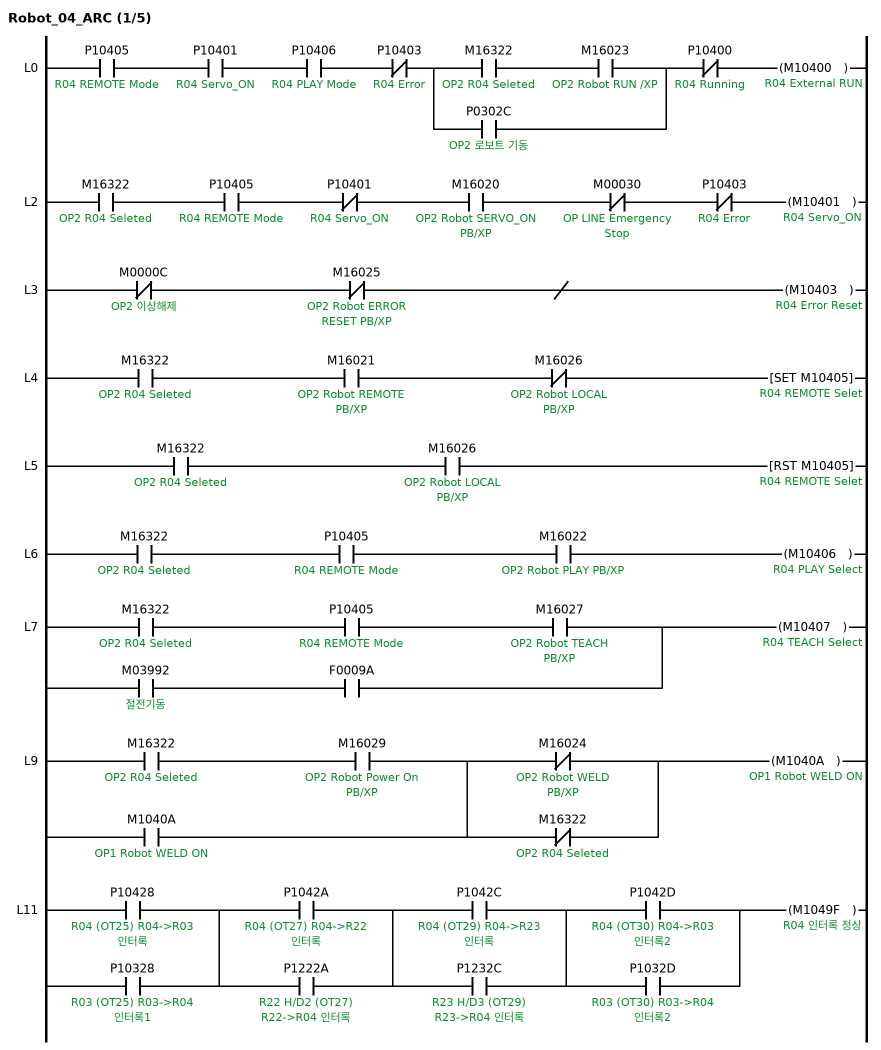
[picture p336: Robot_04_ARC rungs L0-L11]
; L0
LOAD      P10405	// R04 REMOTE Mode
AND       P10401	// R04 Servo_ON
AND       P10406	// R04 PLAY Mode
AND NOT   P10403	// R04 Error
LOAD      M16322	// OP2 R04 Seleted
AND       M16023	// OP2 Robot RUN /XP
OR        P0302C	// OP2 로보트 기동
AND LOAD
AND NOT   P10400	// R04 Running
OUT       M10400	// R04 External RUN
; L2
LOAD      M16322	// OP2 R04 Seleted
AND       P10405	// R04 REMOTE Mode
AND NOT   P10401	// R04 Servo_ON
AND       M16020	// OP2 Robot SERVO_ON PB/XP
AND NOT   M00030	// OP LINE Emergency Stop
AND NOT   P10403	// R04 Error
OUT       M10401	// R04 Servo_ON
; L3
LOAD NOT  M0000C	// OP2 이상해제
AND NOT   M16025	// OP2 Robot ERROR RESET PB/XP
NOT
OUT       M10403	// R04 Error Reset
; L4
LOAD      M16322	// OP2 R04 Seleted
AND       M16021	// OP2 Robot REMOTE PB/XP
AND NOT   M16026	// OP2 Robot LOCAL PB/XP
SET       M10405	// R04 REMOTE Selet
; L5
LOAD      M16322	// OP2 R04 Seleted
AND       M16026	// OP2 Robot LOCAL PB/XP
RST       M10405	// R04 REMOTE Selet
; L6
LOAD      M16322	// OP2 R04 Seleted
AND       P10405	// R04 REMOTE Mode
AND       M16022	// OP2 Robot PLAY PB/XP
OUT       M10406	// R04 PLAY Select
; L7
LOAD      M16322	// OP2 R04 Seleted
AND       P10405	// R04 REMOTE Mode
AND       M16027	// OP2 Robot TEACH PB/XP
LOAD      M03992	// 절전기동
AND       F0009A
OR LOAD
OUT       M10407	// R04 TEACH Select
; L9
LOAD      M16322	// OP2 R04 Seleted
AND       M16029	// OP2 Robot Power On PB/XP
OR        M1040A	// OP1 Robot WELD ON
LOAD NOT  M16024	// OP2 Robot WELD PB/XP
OR NOT    M16322	// OP2 R04 Seleted
AND LOAD
OUT       M1040A	// OP1 Robot WELD ON
; L11
LOAD      P10428	// R04 (OT25) R04->R03 인터록
OR        P10328	// R03 (OT25) R03->R04 인터록1
LOAD      P1042A	// R04 (OT27) R04->R22 인터록
OR        P1222A	// R22 H/D2 (OT27) R22->R04 인터록
AND LOAD
LOAD      P1042C	// R04 (OT29) R04->R23 인터록
OR        P1232C	// R23 H/D3 (OT29) R23->R04 인터록
AND LOAD
LOAD      P1042D	// R04 (OT30) R04->R03 인터록2
OR        P1032D	// R03 (OT30) R03->R04 인터록2
AND LOAD
OUT       M1049F	// R04 인터록 정상

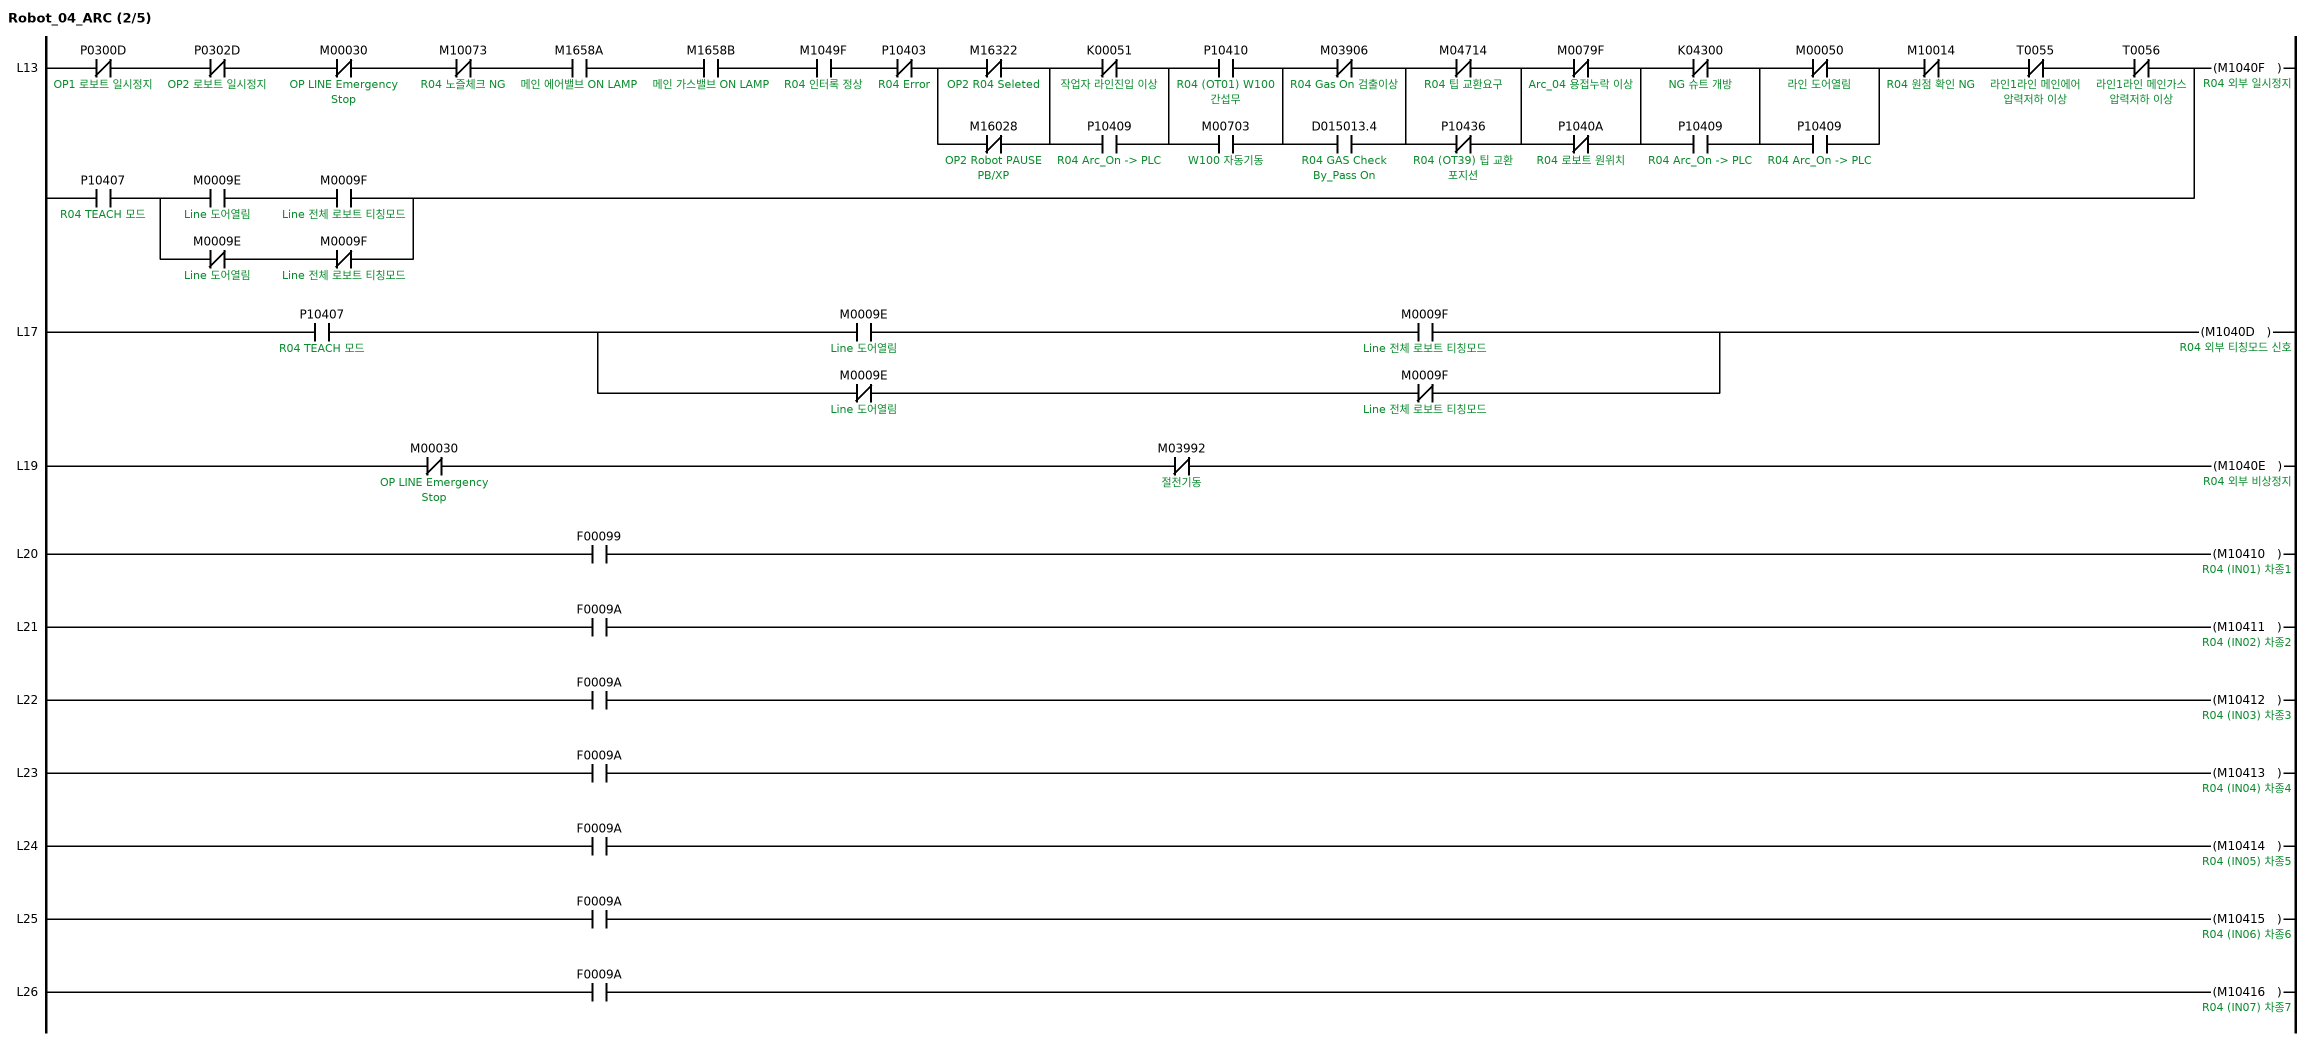
; L13
LOAD NOT  P0300D	// OP1 로보트 일시정지
AND NOT   P0302D	// OP2 로보트 일시정지
AND NOT   M00030	// OP LINE Emergency Stop
AND NOT   M10073	// R04 노즐체크 NG
AND       M1658A	// 메인 에어밸브 ON LAMP
AND       M1658B	// 메인 가스밸브 ON LAMP
AND       M1049F	// R04 인터록 정상
AND NOT   P10403	// R04 Error
LOAD NOT  M16322	// OP2 R04 Seleted
OR NOT    M16028	// OP2 Robot PAUSE PB/XP
AND LOAD
LOAD NOT  K00051	//  작업자 라인진입 이상
OR        P10409	// R04 Arc_On -> PLC
AND LOAD
LOAD      P10410	// R04 (OT01) W100 간섭무
OR        M00703	// W100 자동기동
AND LOAD
LOAD NOT  M03906	// R04 Gas On 검출이상
OR        D015013.4	// R04 GAS Check By_Pass On
AND LOAD
LOAD NOT  M04714	// R04 팁 교환요구
OR NOT    P10436	// R04 (OT39) 팁 교환 포지션
AND LOAD
LOAD NOT  M0079F	// Arc_04 용접누락 이상
OR NOT    P1040A	// R04 로보트 원위치
AND LOAD
LOAD NOT  K04300	// NG 슈트 개방
OR        P10409	// R04 Arc_On -> PLC
AND LOAD
LOAD NOT  M00050	// 라인 도어열림
OR        P10409	// R04 Arc_On -> PLC
AND LOAD
AND NOT   M10014	// R04 원점 확인 NG
AND NOT   T0055	// 라인1라인 메인에어 압력저하 이상
AND NOT   T0056	// 라인1라인 메인가스 압력저하 이상
LOAD      P10407	// R04 TEACH 모드
LOAD      M0009E	// Line 도어열림
AND       M0009F	// Line 전체 로보트 티칭모드
LOAD NOT  M0009E	// Line 도어열림
AND NOT   M0009F	// Line 전체 로보트 티칭모드
OR LOAD
AND LOAD
OR LOAD
OUT       M1040F	// R04 외부 일시정지
; L17
LOAD      P10407	// R04 TEACH 모드
LOAD      M0009E	// Line 도어열림
AND       M0009F	// Line 전체 로보트 티칭모드
LOAD NOT  M0009E	// Line 도어열림
AND NOT   M0009F	// Line 전체 로보트 티칭모드
OR LOAD
AND LOAD
OUT       M1040D	// R04 외부 티칭모드 신호
; L19
LOAD NOT  M00030	// OP LINE Emergency Stop
AND NOT   M03992	// 절전기동
OUT       M1040E	// R04 외부 비상정지 
; L20
LOAD      F00099
OUT       M10410	// R04 (IN01) 차종1
; L21
LOAD      F0009A
OUT       M10411	// R04 (IN02) 차종2
; L22
LOAD      F0009A
OUT       M10412	// R04 (IN03) 차종3
; L23
LOAD      F0009A
OUT       M10413	// R04 (IN04) 차종4
; L24
LOAD      F0009A
OUT       M10414	// R04 (IN05) 차종5
; L25
LOAD      F0009A
OUT       M10415	// R04 (IN06) 차종6
; L26
LOAD      F0009A
OUT       M10416	// R04 (IN07) 차종7

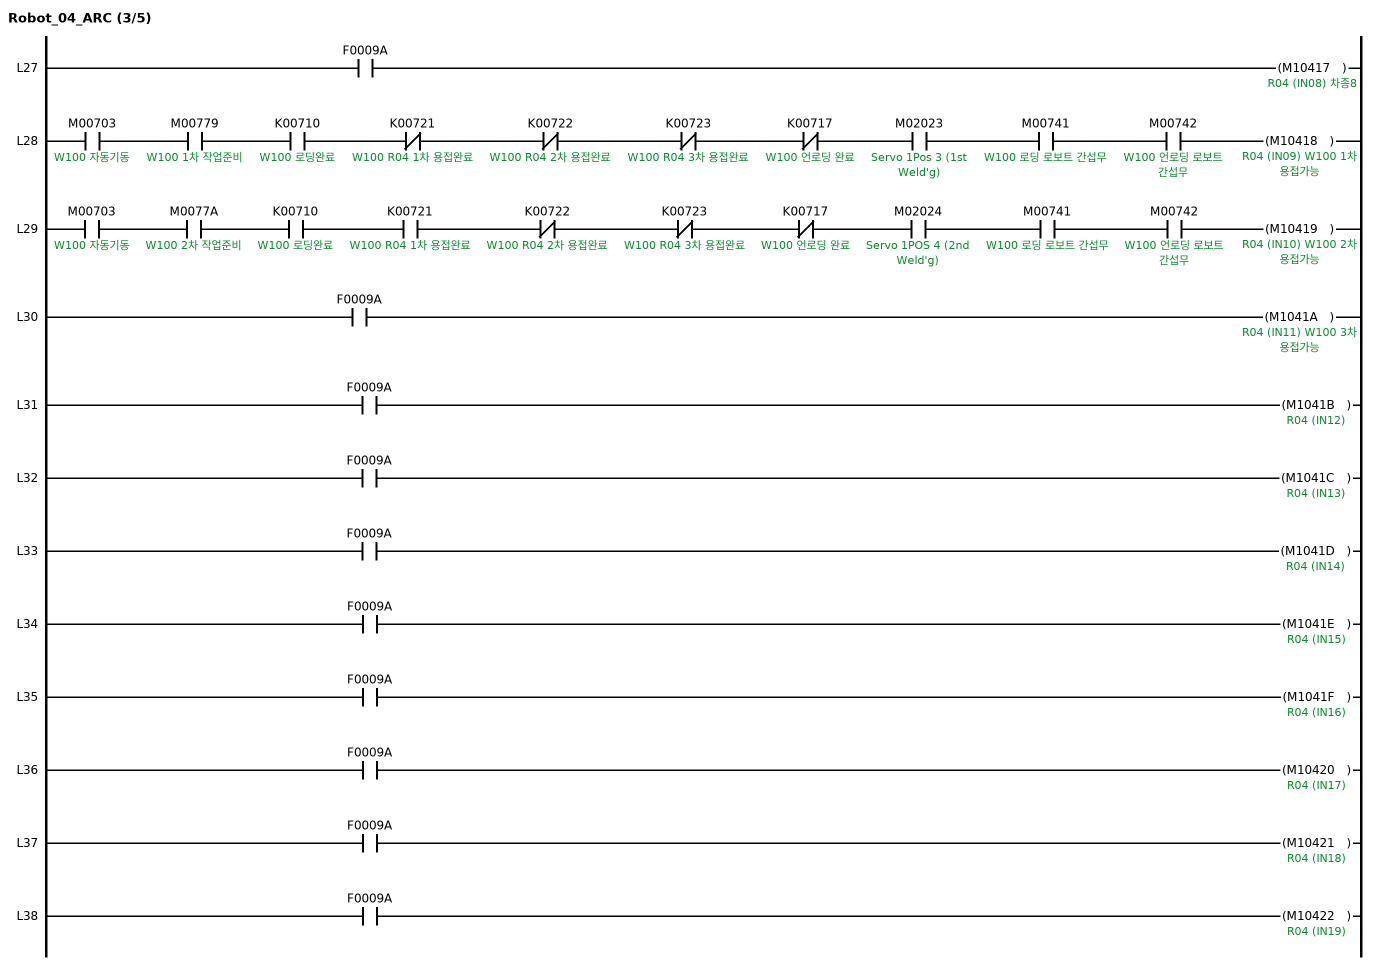
; L27
LOAD      F0009A
OUT       M10417	// R04 (IN08) 차종8
; L28
LOAD      M00703	// W100 자동기동
AND       M00779	// W100 1차 작업준비
AND       K00710	// W100 로딩완료
AND NOT   K00721	// W100 R04 1차 용접완료
AND NOT   K00722	// W100 R04 2차 용접완료
AND NOT   K00723	// W100 R04 3차 용접완료
AND NOT   K00717	// W100 언로딩 완료
AND       M02023	// Servo 1Pos 3 (1st Weld'g)
AND       M00741	// W100 로딩 로보트 간섭무
AND       M00742	// W100 언로딩 로보트 간섭무
OUT       M10418	// R04 (IN09) W100 1차 용접가능
; L29
LOAD      M00703	// W100 자동기동
AND       M0077A	// W100 2차 작업준비
AND       K00710	// W100 로딩완료
AND       K00721	// W100 R04 1차 용접완료
AND NOT   K00722	// W100 R04 2차 용접완료
AND NOT   K00723	// W100 R04 3차 용접완료
AND NOT   K00717	// W100 언로딩 완료
AND       M02024	// Servo 1POS 4 (2nd Weld'g)
AND       M00741	// W100 로딩 로보트 간섭무
AND       M00742	// W100 언로딩 로보트 간섭무
OUT       M10419	// R04 (IN10) W100 2차 용접가능
; L30
LOAD      F0009A
OUT       M1041A	// R04 (IN11) W100 3차 용접가능
; L31
LOAD      F0009A
OUT       M1041B	// R04 (IN12)
; L32
LOAD      F0009A
OUT       M1041C	// R04 (IN13)
; L33
LOAD      F0009A
OUT       M1041D	// R04 (IN14)
; L34
LOAD      F0009A
OUT       M1041E	// R04 (IN15)
; L35
LOAD      F0009A
OUT       M1041F	// R04 (IN16)
; L36
LOAD      F0009A
OUT       M10420	// R04 (IN17)
; L37
LOAD      F0009A
OUT       M10421	// R04 (IN18)
; L38
LOAD      F0009A
OUT       M10422	// R04 (IN19)

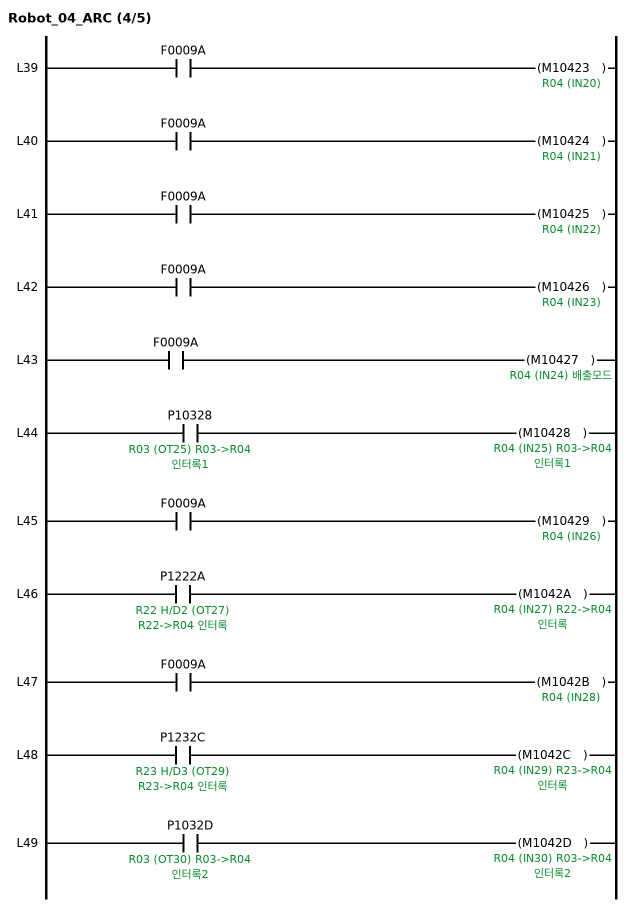
; L39
LOAD      F0009A
OUT       M10423	// R04 (IN20)
; L40
LOAD      F0009A
OUT       M10424	// R04 (IN21)
; L41
LOAD      F0009A
OUT       M10425	// R04 (IN22)
; L42
LOAD      F0009A
OUT       M10426	// R04 (IN23)
; L43
LOAD      F0009A
OUT       M10427	// R04 (IN24) 배출모드
; L44
LOAD      P10328	// R03 (OT25) R03->R04 인터록1
OUT       M10428	// R04 (IN25) R03->R04 인터록1
; L45
LOAD      F0009A
OUT       M10429	// R04 (IN26)
; L46
LOAD      P1222A	// R22 H/D2 (OT27) R22->R04 인터록
OUT       M1042A	// R04 (IN27) R22->R04 인터록
; L47
LOAD      F0009A
OUT       M1042B	// R04 (IN28)
; L48
LOAD      P1232C	// R23 H/D3 (OT29) R23->R04 인터록
OUT       M1042C	// R04 (IN29) R23->R04 인터록
; L49
LOAD      P1032D	// R03 (OT30) R03->R04 인터록2
OUT       M1042D	// R04 (IN30) R03->R04 인터록2

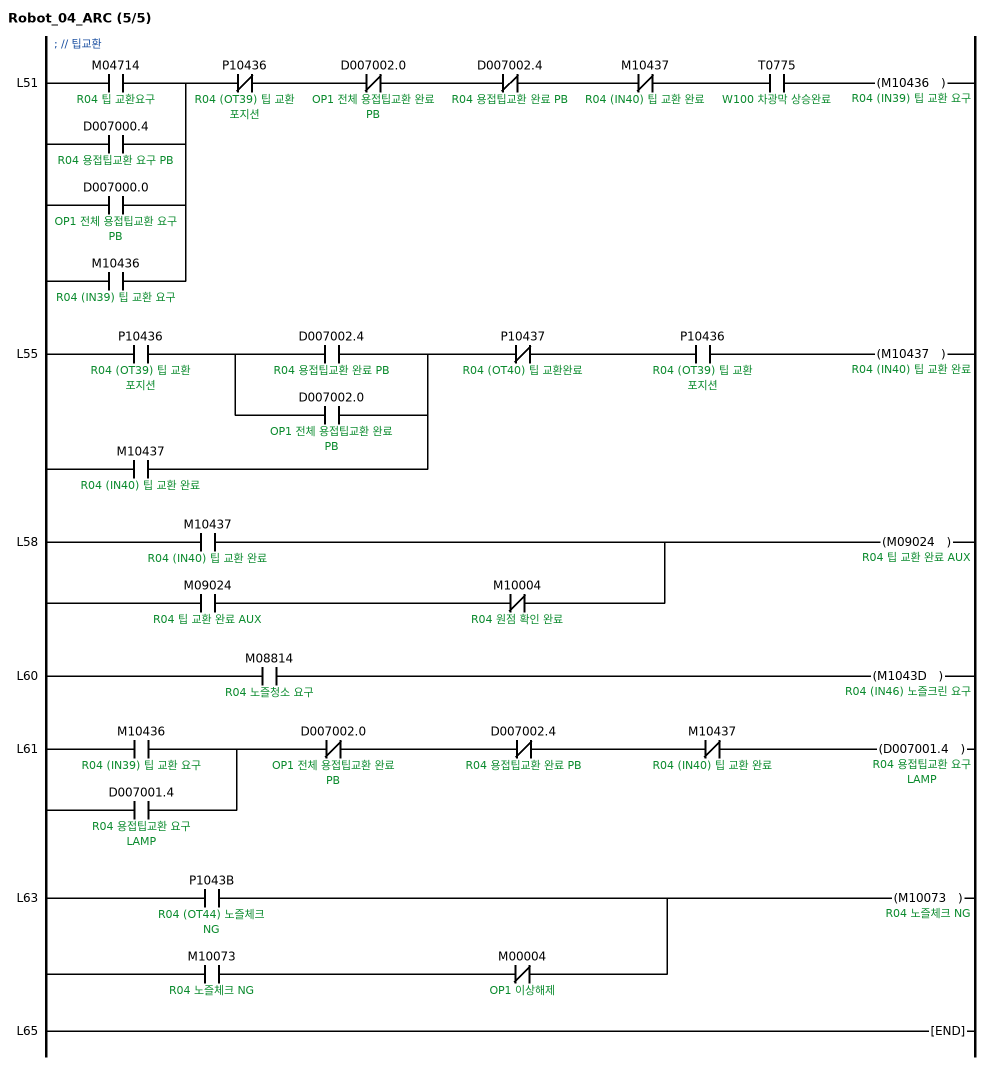
//  // 팁교환
; L51
LOAD      M04714	// R04 팁 교환요구
OR        D007000.4	// R04 용접팁교환 요구 PB
OR        D007000.0	// OP1 전체 용접팁교환 요구 PB
OR        M10436	// R04 (IN39) 팁 교환 요구
AND NOT   P10436	// R04 (OT39) 팁 교환 포지션
AND NOT   D007002.0	// OP1 전체 용접팁교환 완료 PB
AND NOT   D007002.4	// R04 용접팁교환 완료 PB
AND NOT   M10437	// R04 (IN40) 팁 교환 완료
AND       T0775	// W100 차광막 상승완료
OUT       M10436	// R04 (IN39) 팁 교환 요구
; L55
LOAD      P10436	// R04 (OT39) 팁 교환 포지션
LOAD      D007002.4	// R04 용접팁교환 완료 PB
OR        D007002.0	// OP1 전체 용접팁교환 완료 PB
AND LOAD
OR        M10437	// R04 (IN40) 팁 교환 완료
AND NOT   P10437	// R04 (OT40) 팁 교환완료
AND       P10436	// R04 (OT39) 팁 교환 포지션
OUT       M10437	// R04 (IN40) 팁 교환 완료
; L58
LOAD      M10437	// R04 (IN40) 팁 교환 완료
LOAD      M09024	// R04 팁 교환 완료 AUX
AND NOT   M10004	// R04 원점 확인 완료
OR LOAD
OUT       M09024	// R04 팁 교환 완료 AUX
; L60
LOAD      M08814	// R04 노즐청소 요구
OUT       M1043D	// R04 (IN46) 노즐크린 요구
; L61
LOAD      M10436	// R04 (IN39) 팁 교환 요구
OR        D007001.4	// R04 용접팁교환 요구 LAMP
AND NOT   D007002.0	// OP1 전체 용접팁교환 완료 PB
AND NOT   D007002.4	// R04 용접팁교환 완료 PB
AND NOT   M10437	// R04 (IN40) 팁 교환 완료
OUT       D007001.4	// R04 용접팁교환 요구 LAMP
; L63
LOAD      P1043B	// R04 (OT44) 노즐체크 NG
LOAD      M10073	// R04 노즐체크 NG
AND NOT   M00004	// OP1 이상해제
OR LOAD
OUT       M10073	// R04 노즐체크 NG
; L65
END

PROGRAM Robot_05_ARC (task: 스캔 프로그램)

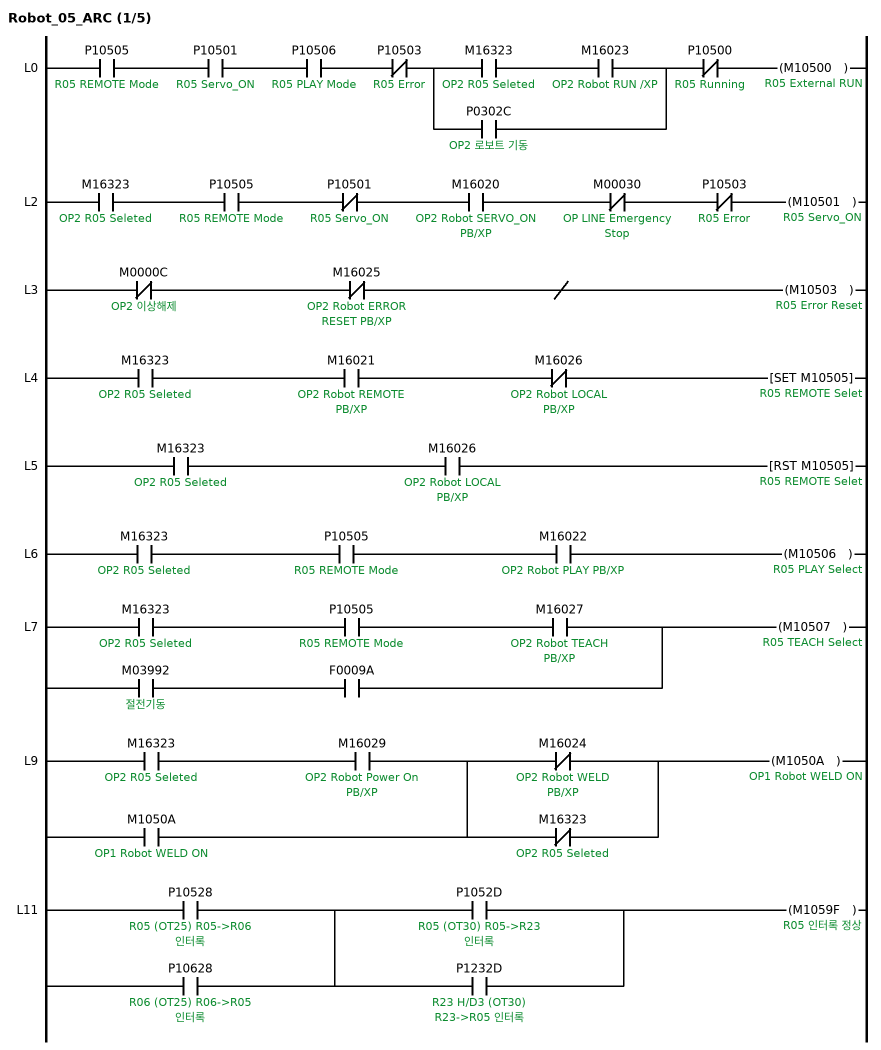
; L0
LOAD      P10505	// R05 REMOTE Mode
AND       P10501	// R05 Servo_ON
AND       P10506	// R05 PLAY Mode
AND NOT   P10503	// R05 Error
LOAD      M16323	// OP2 R05 Seleted
AND       M16023	// OP2 Robot RUN /XP
OR        P0302C	// OP2 로보트 기동
AND LOAD
AND NOT   P10500	// R05 Running
OUT       M10500	// R05 External RUN
; L2
LOAD      M16323	// OP2 R05 Seleted
AND       P10505	// R05 REMOTE Mode
AND NOT   P10501	// R05 Servo_ON
AND       M16020	// OP2 Robot SERVO_ON PB/XP
AND NOT   M00030	// OP LINE Emergency Stop
AND NOT   P10503	// R05 Error
OUT       M10501	// R05 Servo_ON
; L3
LOAD NOT  M0000C	// OP2 이상해제
AND NOT   M16025	// OP2 Robot ERROR RESET PB/XP
NOT
OUT       M10503	// R05 Error Reset
; L4
LOAD      M16323	// OP2 R05 Seleted
AND       M16021	// OP2 Robot REMOTE PB/XP
AND NOT   M16026	// OP2 Robot LOCAL PB/XP
SET       M10505	// R05 REMOTE Selet
; L5
LOAD      M16323	// OP2 R05 Seleted
AND       M16026	// OP2 Robot LOCAL PB/XP
RST       M10505	// R05 REMOTE Selet
; L6
LOAD      M16323	// OP2 R05 Seleted
AND       P10505	// R05 REMOTE Mode
AND       M16022	// OP2 Robot PLAY PB/XP
OUT       M10506	// R05 PLAY Select
; L7
LOAD      M16323	// OP2 R05 Seleted
AND       P10505	// R05 REMOTE Mode
AND       M16027	// OP2 Robot TEACH PB/XP
LOAD      M03992	// 절전기동
AND       F0009A
OR LOAD
OUT       M10507	// R05 TEACH Select
; L9
LOAD      M16323	// OP2 R05 Seleted
AND       M16029	// OP2 Robot Power On PB/XP
OR        M1050A	// OP1 Robot WELD ON
LOAD NOT  M16024	// OP2 Robot WELD PB/XP
OR NOT    M16323	// OP2 R05 Seleted
AND LOAD
OUT       M1050A	// OP1 Robot WELD ON
; L11
LOAD      P10528	// R05 (OT25) R05->R06 인터록
OR        P10628	// R06 (OT25) R06->R05 인터록
LOAD      P1052D	// R05 (OT30) R05->R23 인터록
OR        P1232D	// R23 H/D3 (OT30) R23->R05 인터록
AND LOAD
OUT       M1059F	// R05 인터록 정상

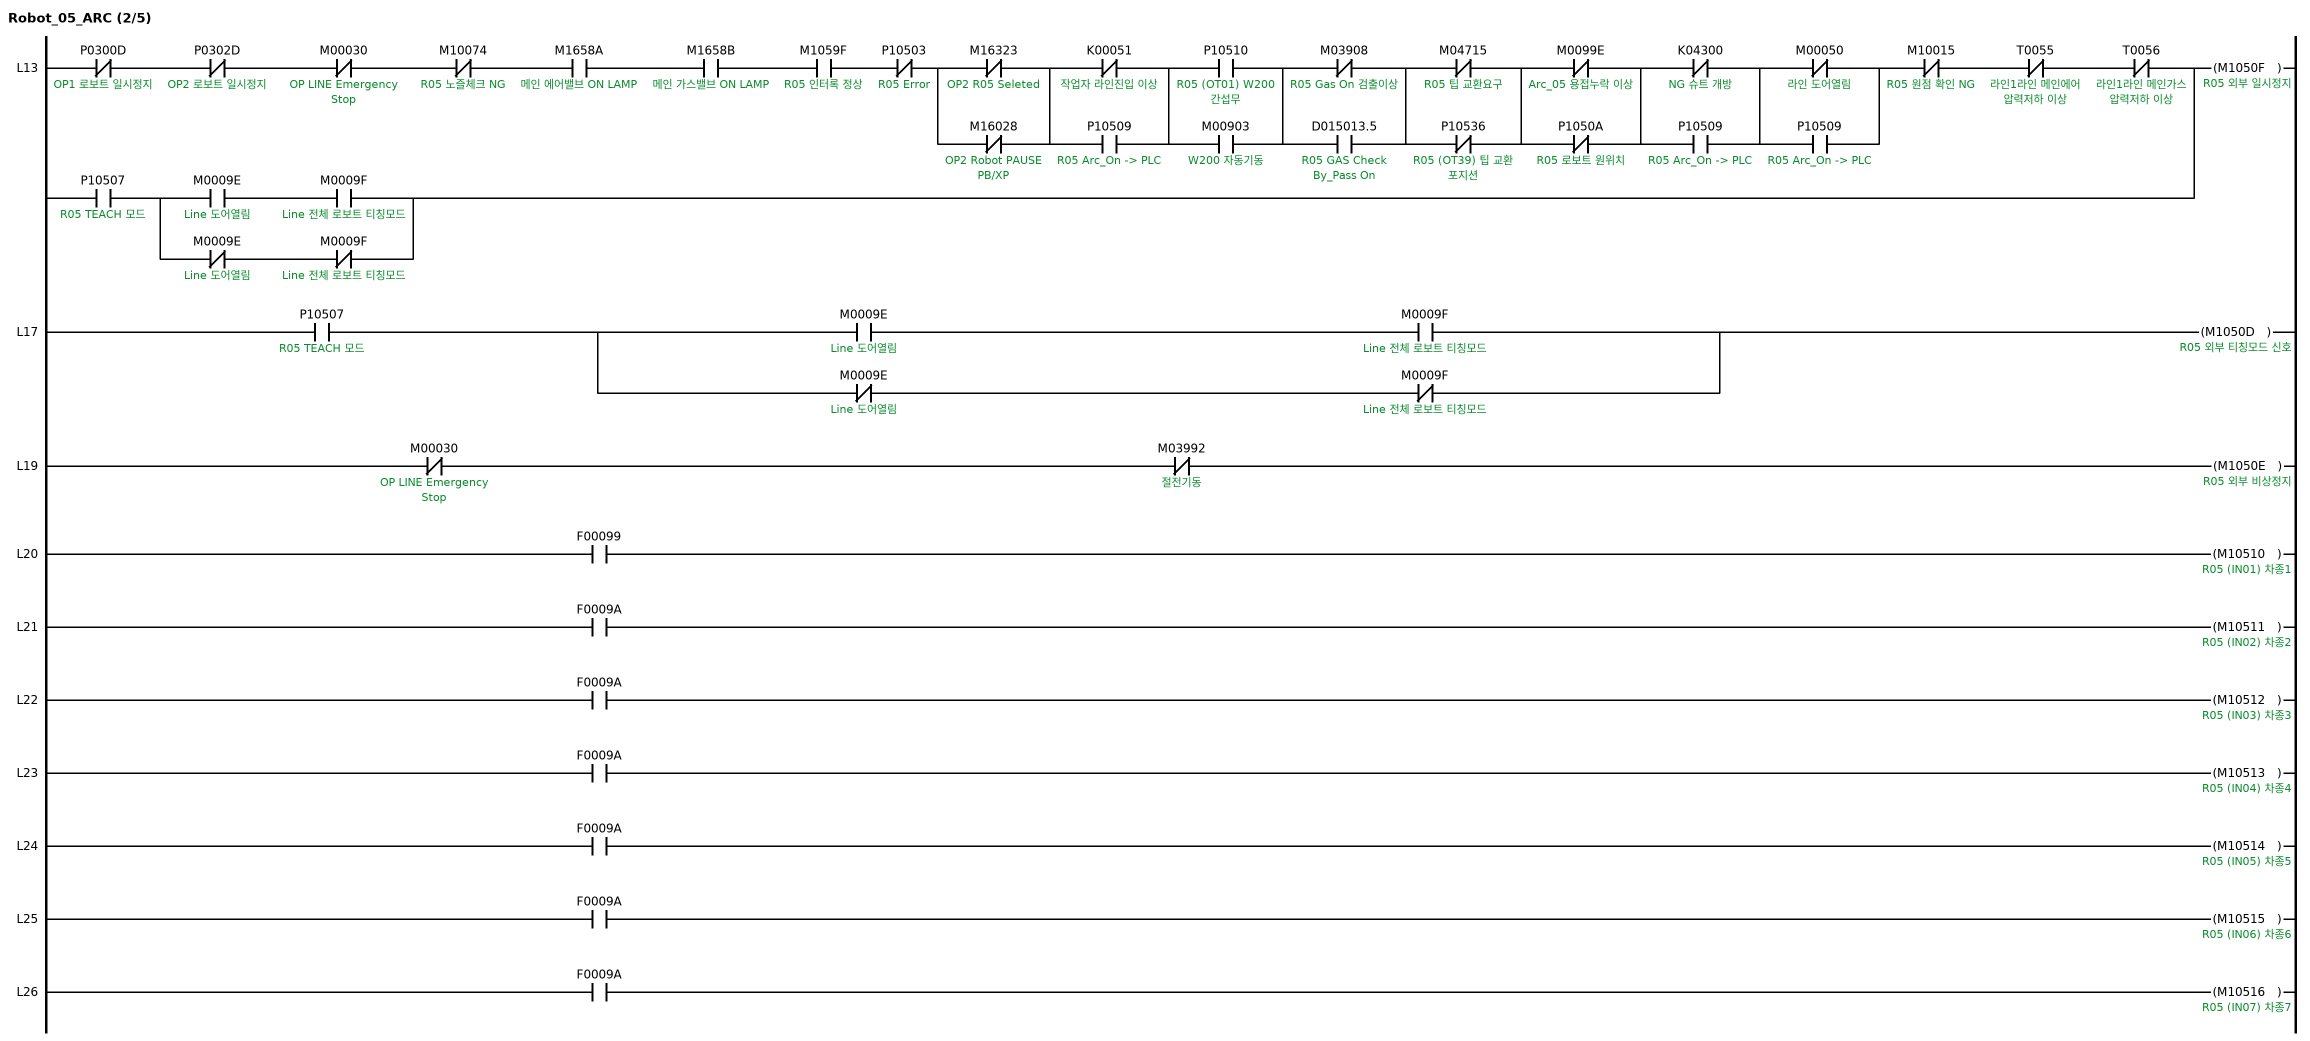
; L13
LOAD NOT  P0300D	// OP1 로보트 일시정지
AND NOT   P0302D	// OP2 로보트 일시정지
AND NOT   M00030	// OP LINE Emergency Stop
AND NOT   M10074	// R05 노즐체크 NG
AND       M1658A	// 메인 에어밸브 ON LAMP
AND       M1658B	// 메인 가스밸브 ON LAMP
AND       M1059F	// R05 인터록 정상
AND NOT   P10503	// R05 Error
LOAD NOT  M16323	// OP2 R05 Seleted
OR NOT    M16028	// OP2 Robot PAUSE PB/XP
AND LOAD
LOAD NOT  K00051	//  작업자 라인진입 이상
OR        P10509	// R05 Arc_On -> PLC
AND LOAD
LOAD      P10510	// R05 (OT01) W200 간섭무
OR        M00903	// W200 자동기동
AND LOAD
LOAD NOT  M03908	// R05 Gas On 검출이상
OR        D015013.5	// R05 GAS Check By_Pass On
AND LOAD
LOAD NOT  M04715	// R05 팁 교환요구
OR NOT    P10536	// R05 (OT39) 팁 교환 포지션
AND LOAD
LOAD NOT  M0099E	// Arc_05 용접누락 이상
OR NOT    P1050A	// R05 로보트 원위치
AND LOAD
LOAD NOT  K04300	// NG 슈트 개방
OR        P10509	// R05 Arc_On -> PLC
AND LOAD
LOAD NOT  M00050	// 라인 도어열림
OR        P10509	// R05 Arc_On -> PLC
AND LOAD
AND NOT   M10015	// R05 원점 확인 NG
AND NOT   T0055	// 라인1라인 메인에어 압력저하 이상
AND NOT   T0056	// 라인1라인 메인가스 압력저하 이상
LOAD      P10507	// R05 TEACH 모드
LOAD      M0009E	// Line 도어열림
AND       M0009F	// Line 전체 로보트 티칭모드
LOAD NOT  M0009E	// Line 도어열림
AND NOT   M0009F	// Line 전체 로보트 티칭모드
OR LOAD
AND LOAD
OR LOAD
OUT       M1050F	// R05 외부 일시정지
; L17
LOAD      P10507	// R05 TEACH 모드
LOAD      M0009E	// Line 도어열림
AND       M0009F	// Line 전체 로보트 티칭모드
LOAD NOT  M0009E	// Line 도어열림
AND NOT   M0009F	// Line 전체 로보트 티칭모드
OR LOAD
AND LOAD
OUT       M1050D	// R05 외부 티칭모드 신호
; L19
LOAD NOT  M00030	// OP LINE Emergency Stop
AND NOT   M03992	// 절전기동
OUT       M1050E	// R05 외부 비상정지 
; L20
LOAD      F00099
OUT       M10510	// R05 (IN01) 차종1
; L21
LOAD      F0009A
OUT       M10511	// R05 (IN02) 차종2
; L22
LOAD      F0009A
OUT       M10512	// R05 (IN03) 차종3
; L23
LOAD      F0009A
OUT       M10513	// R05 (IN04) 차종4
; L24
LOAD      F0009A
OUT       M10514	// R05 (IN05) 차종5
; L25
LOAD      F0009A
OUT       M10515	// R05 (IN06) 차종6
; L26
LOAD      F0009A
OUT       M10516	// R05 (IN07) 차종7

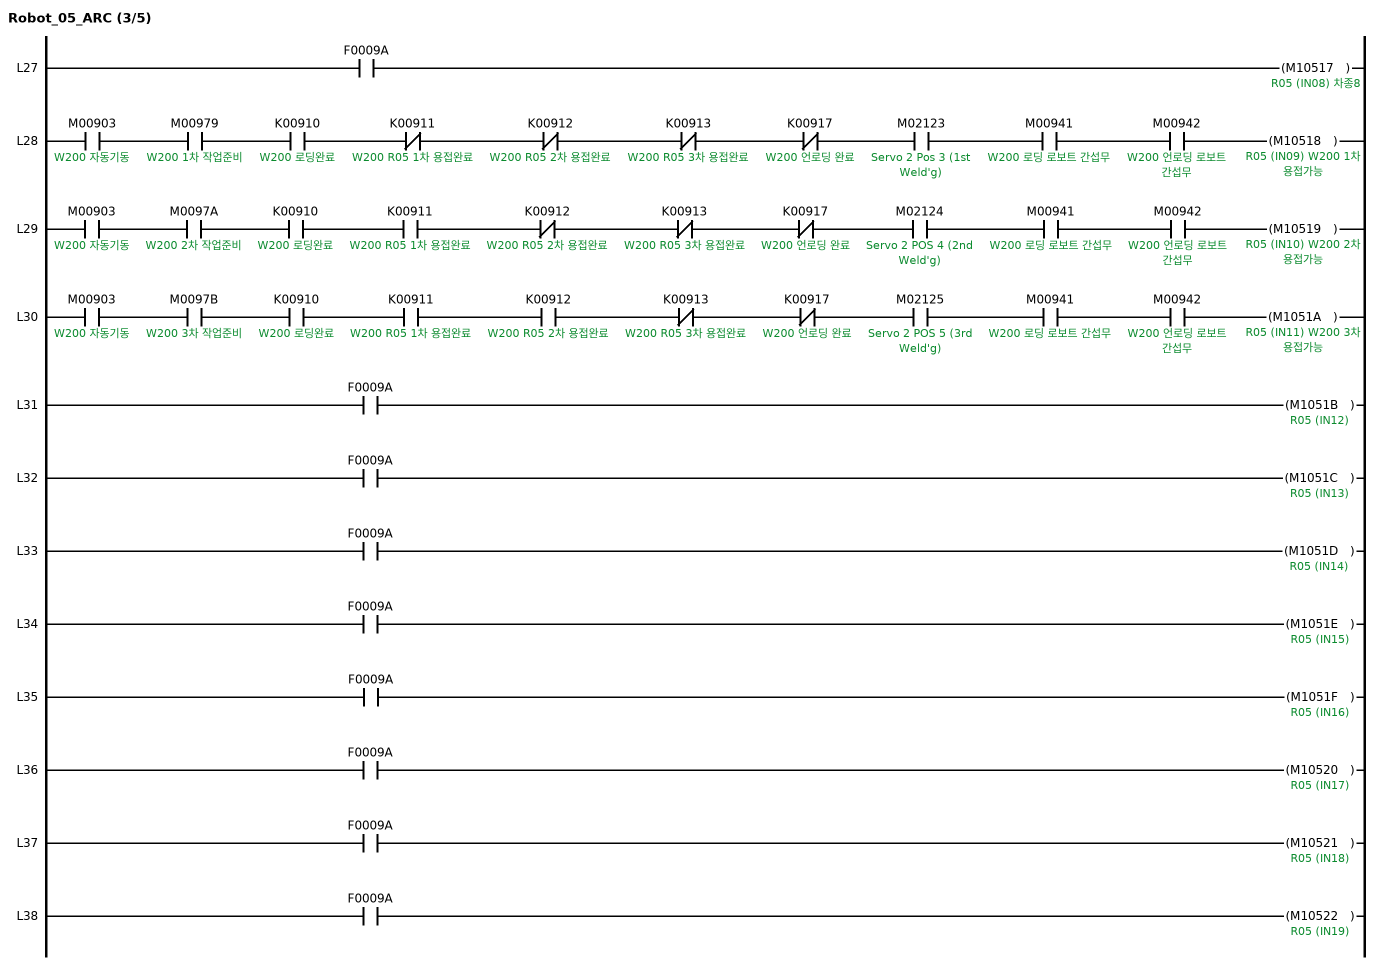
; L27
LOAD      F0009A
OUT       M10517	// R05 (IN08) 차종8
; L28
LOAD      M00903	// W200 자동기동
AND       M00979	// W200 1차 작업준비
AND       K00910	// W200 로딩완료
AND NOT   K00911	// W200 R05 1차 용접완료
AND NOT   K00912	// W200 R05 2차 용접완료
AND NOT   K00913	// W200 R05 3차 용접완료
AND NOT   K00917	// W200 언로딩 완료
AND       M02123	// Servo 2 Pos 3 (1st Weld'g)
AND       M00941	// W200 로딩 로보트 간섭무
AND       M00942	// W200 언로딩 로보트 간섭무
OUT       M10518	// R05 (IN09) W200 1차 용접가능
; L29
LOAD      M00903	// W200 자동기동
AND       M0097A	// W200 2차 작업준비
AND       K00910	// W200 로딩완료
AND       K00911	// W200 R05 1차 용접완료
AND NOT   K00912	// W200 R05 2차 용접완료
AND NOT   K00913	// W200 R05 3차 용접완료
AND NOT   K00917	// W200 언로딩 완료
AND       M02124	// Servo 2 POS 4 (2nd Weld'g)
AND       M00941	// W200 로딩 로보트 간섭무
AND       M00942	// W200 언로딩 로보트 간섭무
OUT       M10519	// R05 (IN10) W200 2차 용접가능
; L30
LOAD      M00903	// W200 자동기동
AND       M0097B	// W200 3차 작업준비
AND       K00910	// W200 로딩완료
AND       K00911	// W200 R05 1차 용접완료
AND       K00912	// W200 R05 2차 용접완료
AND NOT   K00913	// W200 R05 3차 용접완료
AND NOT   K00917	// W200 언로딩 완료
AND       M02125	// Servo 2 POS 5 (3rd Weld'g)
AND       M00941	// W200 로딩 로보트 간섭무
AND       M00942	// W200 언로딩 로보트 간섭무
OUT       M1051A	// R05 (IN11) W200 3차 용접가능
; L31
LOAD      F0009A
OUT       M1051B	// R05 (IN12)
; L32
LOAD      F0009A
OUT       M1051C	// R05 (IN13)
; L33
LOAD      F0009A
OUT       M1051D	// R05 (IN14)
; L34
LOAD      F0009A
OUT       M1051E	// R05 (IN15)
; L35
LOAD      F0009A
OUT       M1051F	// R05 (IN16)
; L36
LOAD      F0009A
OUT       M10520	// R05 (IN17)
; L37
LOAD      F0009A
OUT       M10521	// R05 (IN18)
; L38
LOAD      F0009A
OUT       M10522	// R05 (IN19)

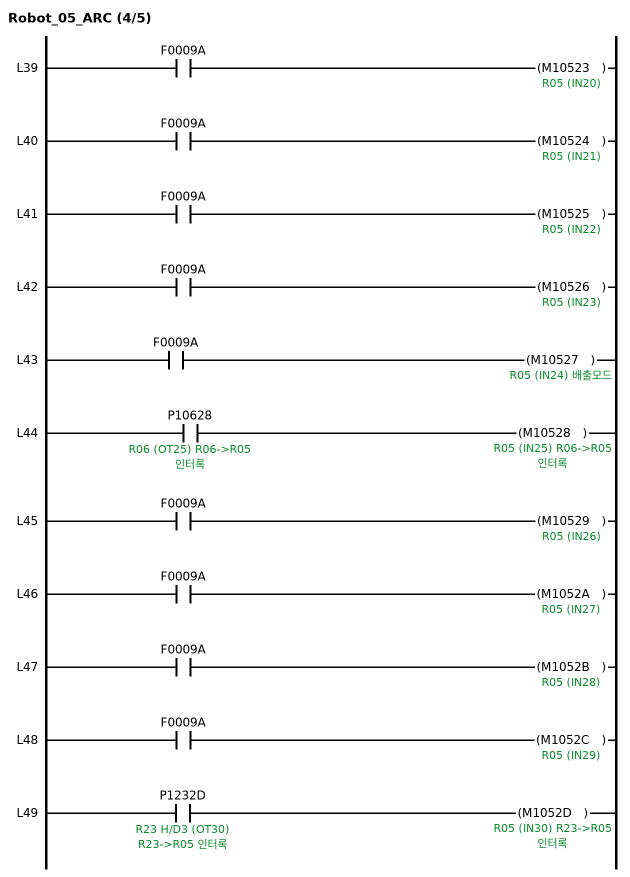
; L39
LOAD      F0009A
OUT       M10523	// R05 (IN20)
; L40
LOAD      F0009A
OUT       M10524	// R05 (IN21)
; L41
LOAD      F0009A
OUT       M10525	// R05 (IN22)
; L42
LOAD      F0009A
OUT       M10526	// R05 (IN23)
; L43
LOAD      F0009A
OUT       M10527	// R05 (IN24) 배출모드
; L44
LOAD      P10628	// R06 (OT25) R06->R05 인터록
OUT       M10528	// R05 (IN25) R06->R05 인터록
; L45
LOAD      F0009A
OUT       M10529	// R05 (IN26)
; L46
LOAD      F0009A
OUT       M1052A	// R05 (IN27)
; L47
LOAD      F0009A
OUT       M1052B	// R05 (IN28)
; L48
LOAD      F0009A
OUT       M1052C	// R05 (IN29)
; L49
LOAD      P1232D	// R23 H/D3 (OT30) R23->R05 인터록
OUT       M1052D	// R05 (IN30) R23->R05 인터록

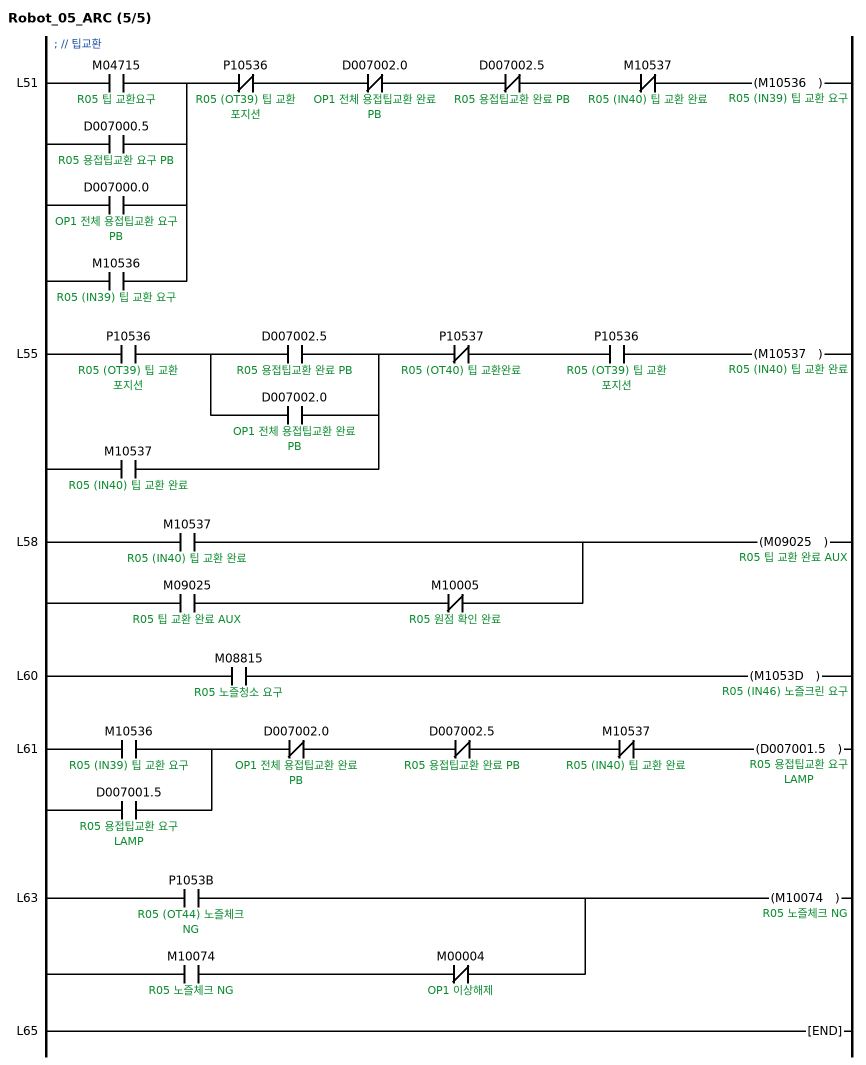
//  // 팁교환
; L51
LOAD      M04715	// R05 팁 교환요구
OR        D007000.5	// R05 용접팁교환 요구 PB
OR        D007000.0	// OP1 전체 용접팁교환 요구 PB
OR        M10536	// R05 (IN39) 팁 교환 요구
AND NOT   P10536	// R05 (OT39) 팁 교환 포지션
AND NOT   D007002.0	// OP1 전체 용접팁교환 완료 PB
AND NOT   D007002.5	// R05 용접팁교환 완료 PB
AND NOT   M10537	// R05 (IN40) 팁 교환 완료
OUT       M10536	// R05 (IN39) 팁 교환 요구
; L55
LOAD      P10536	// R05 (OT39) 팁 교환 포지션
LOAD      D007002.5	// R05 용접팁교환 완료 PB
OR        D007002.0	// OP1 전체 용접팁교환 완료 PB
AND LOAD
OR        M10537	// R05 (IN40) 팁 교환 완료
AND NOT   P10537	// R05 (OT40) 팁 교환완료
AND       P10536	// R05 (OT39) 팁 교환 포지션
OUT       M10537	// R05 (IN40) 팁 교환 완료
; L58
LOAD      M10537	// R05 (IN40) 팁 교환 완료
LOAD      M09025	// R05 팁 교환 완료 AUX
AND NOT   M10005	// R05 원점 확인 완료
OR LOAD
OUT       M09025	// R05 팁 교환 완료 AUX
; L60
LOAD      M08815	// R05 노즐청소 요구
OUT       M1053D	// R05 (IN46) 노즐크린 요구
; L61
LOAD      M10536	// R05 (IN39) 팁 교환 요구
OR        D007001.5	// R05 용접팁교환 요구 LAMP
AND NOT   D007002.0	// OP1 전체 용접팁교환 완료 PB
AND NOT   D007002.5	// R05 용접팁교환 완료 PB
AND NOT   M10537	// R05 (IN40) 팁 교환 완료
OUT       D007001.5	// R05 용접팁교환 요구 LAMP
; L63
LOAD      P1053B	// R05 (OT44) 노즐체크 NG
LOAD      M10074	// R05 노즐체크 NG
AND NOT   M00004	// OP1 이상해제
OR LOAD
OUT       M10074	// R05 노즐체크 NG
; L65
END

PROGRAM Robot_06_ARC (task: 스캔 프로그램)

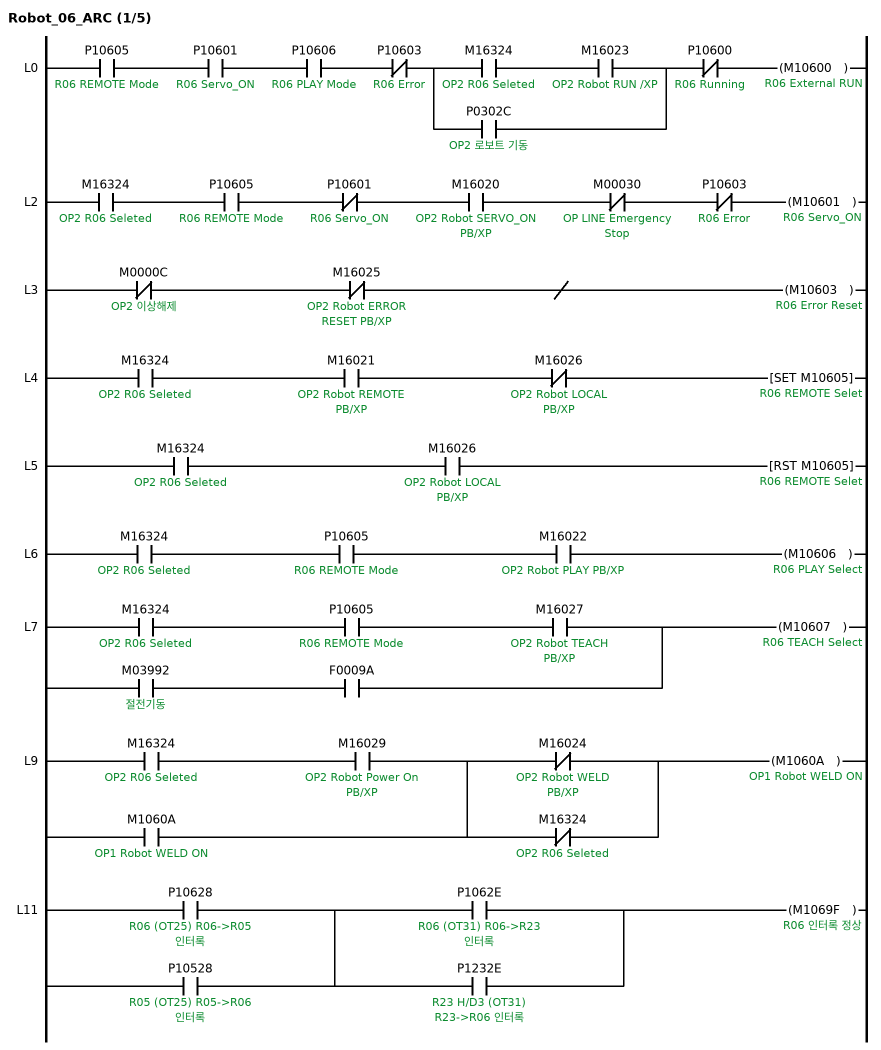
; L0
LOAD      P10605	// R06 REMOTE Mode
AND       P10601	// R06 Servo_ON
AND       P10606	// R06 PLAY Mode
AND NOT   P10603	// R06 Error
LOAD      M16324	// OP2 R06 Seleted
AND       M16023	// OP2 Robot RUN /XP
OR        P0302C	// OP2 로보트 기동
AND LOAD
AND NOT   P10600	// R06 Running
OUT       M10600	// R06 External RUN
; L2
LOAD      M16324	// OP2 R06 Seleted
AND       P10605	// R06 REMOTE Mode
AND NOT   P10601	// R06 Servo_ON
AND       M16020	// OP2 Robot SERVO_ON PB/XP
AND NOT   M00030	// OP LINE Emergency Stop
AND NOT   P10603	// R06 Error
OUT       M10601	// R06 Servo_ON
; L3
LOAD NOT  M0000C	// OP2 이상해제
AND NOT   M16025	// OP2 Robot ERROR RESET PB/XP
NOT
OUT       M10603	// R06 Error Reset
; L4
LOAD      M16324	// OP2 R06 Seleted
AND       M16021	// OP2 Robot REMOTE PB/XP
AND NOT   M16026	// OP2 Robot LOCAL PB/XP
SET       M10605	// R06 REMOTE Selet
; L5
LOAD      M16324	// OP2 R06 Seleted
AND       M16026	// OP2 Robot LOCAL PB/XP
RST       M10605	// R06 REMOTE Selet
; L6
LOAD      M16324	// OP2 R06 Seleted
AND       P10605	// R06 REMOTE Mode
AND       M16022	// OP2 Robot PLAY PB/XP
OUT       M10606	// R06 PLAY Select
; L7
LOAD      M16324	// OP2 R06 Seleted
AND       P10605	// R06 REMOTE Mode
AND       M16027	// OP2 Robot TEACH PB/XP
LOAD      M03992	// 절전기동
AND       F0009A
OR LOAD
OUT       M10607	// R06 TEACH Select
; L9
LOAD      M16324	// OP2 R06 Seleted
AND       M16029	// OP2 Robot Power On PB/XP
OR        M1060A	// OP1 Robot WELD ON
LOAD NOT  M16024	// OP2 Robot WELD PB/XP
OR NOT    M16324	// OP2 R06 Seleted
AND LOAD
OUT       M1060A	// OP1 Robot WELD ON
; L11
LOAD      P10628	// R06 (OT25) R06->R05 인터록
OR        P10528	// R05 (OT25) R05->R06 인터록
LOAD      P1062E	// R06 (OT31) R06->R23 인터록
OR        P1232E	// R23 H/D3 (OT31) R23->R06 인터록
AND LOAD
OUT       M1069F	// R06 인터록 정상

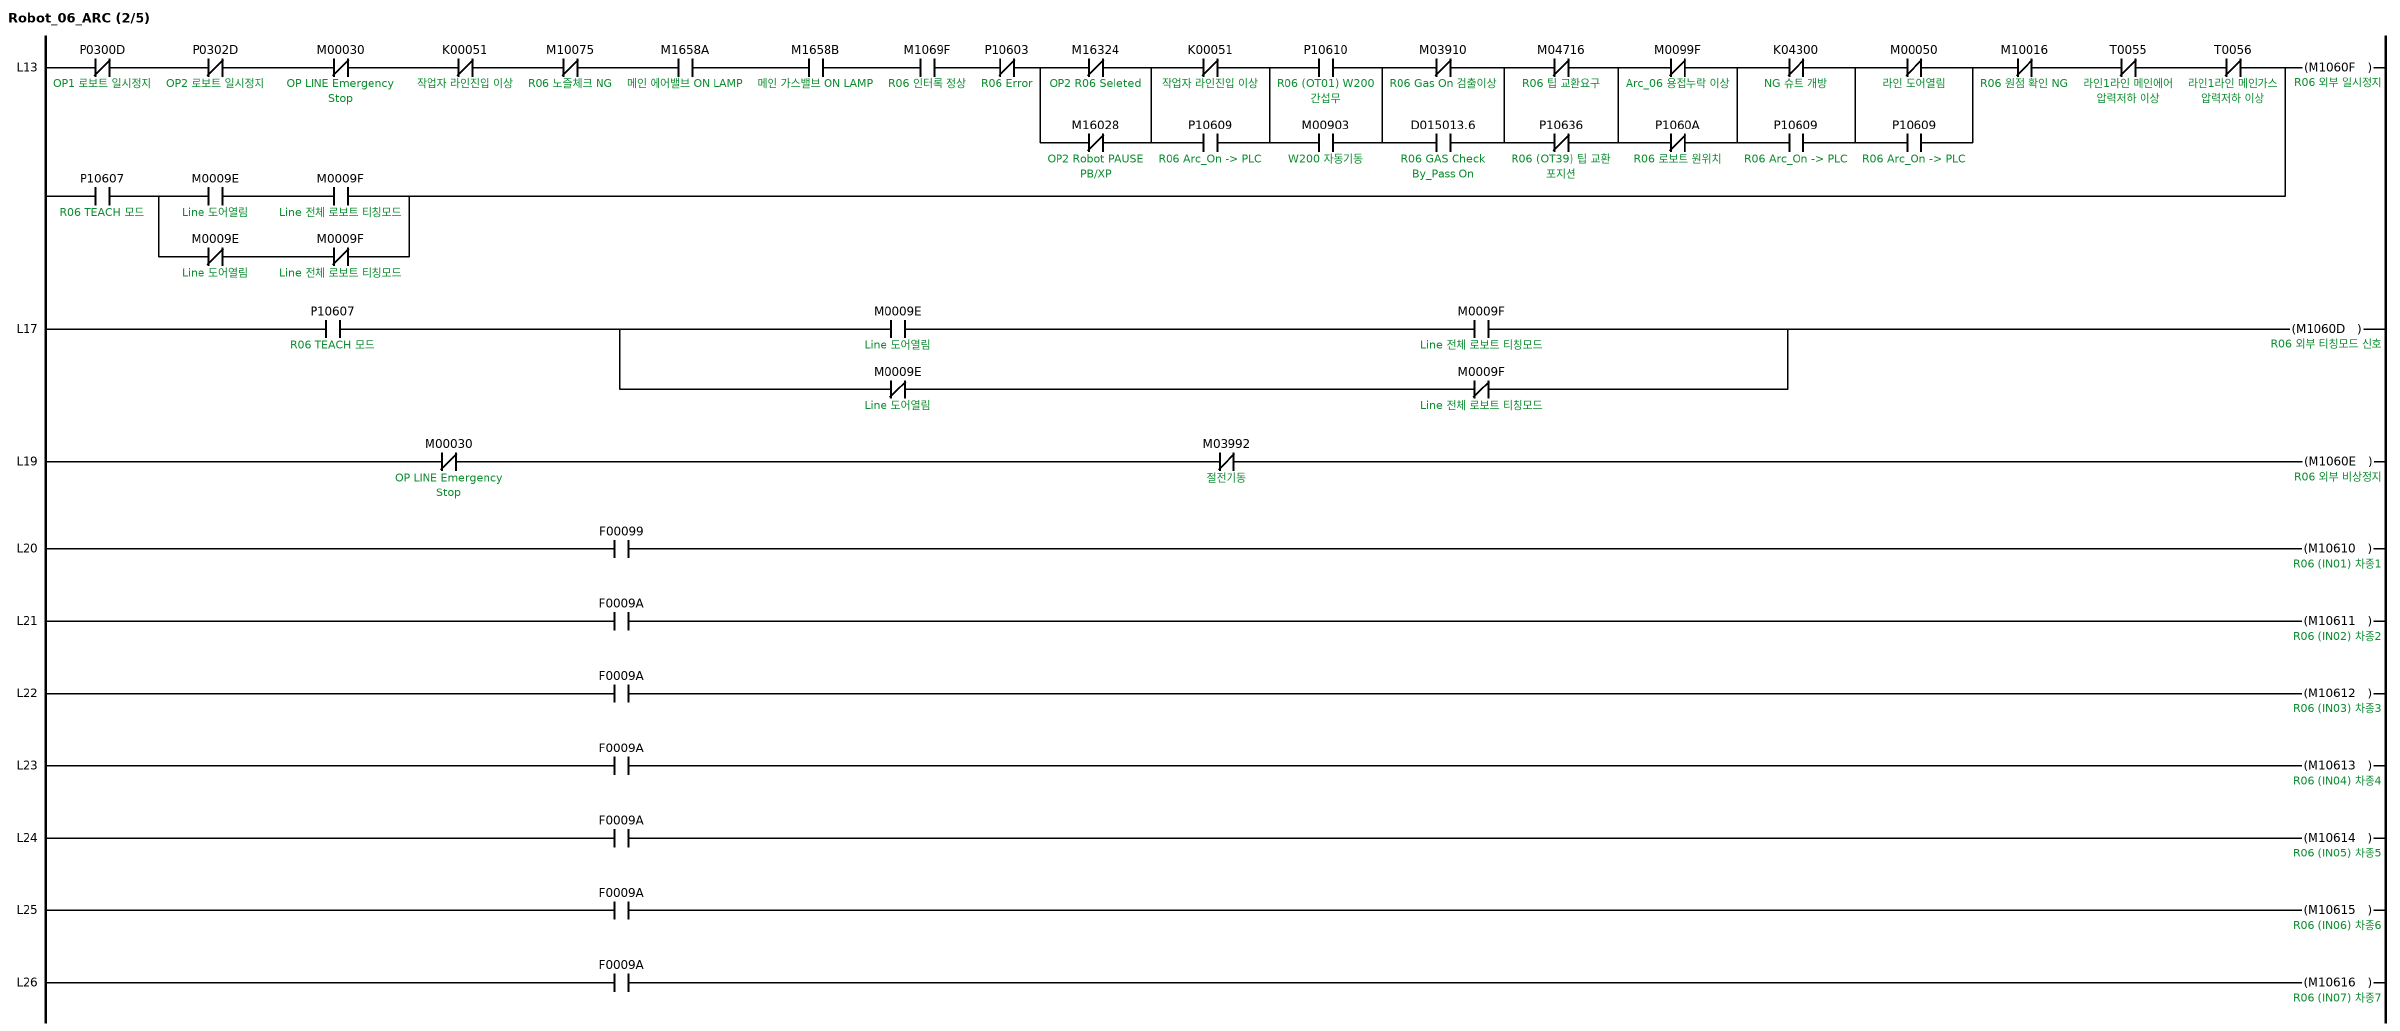
; L13
LOAD NOT  P0300D	// OP1 로보트 일시정지
AND NOT   P0302D	// OP2 로보트 일시정지
AND NOT   M00030	// OP LINE Emergency Stop
AND NOT   K00051	//  작업자 라인진입 이상
AND NOT   M10075	// R06 노즐체크 NG
AND       M1658A	// 메인 에어밸브 ON LAMP
AND       M1658B	// 메인 가스밸브 ON LAMP
AND       M1069F	// R06 인터록 정상
AND NOT   P10603	// R06 Error
LOAD NOT  M16324	// OP2 R06 Seleted
OR NOT    M16028	// OP2 Robot PAUSE PB/XP
AND LOAD
LOAD NOT  K00051	//  작업자 라인진입 이상
OR        P10609	// R06 Arc_On -> PLC
AND LOAD
LOAD      P10610	// R06 (OT01) W200 간섭무
OR        M00903	// W200 자동기동
AND LOAD
LOAD NOT  M03910	// R06 Gas On 검출이상
OR        D015013.6	// R06 GAS Check By_Pass On
AND LOAD
LOAD NOT  M04716	// R06 팁 교환요구
OR NOT    P10636	// R06 (OT39) 팁 교환 포지션
AND LOAD
LOAD NOT  M0099F	// Arc_06 용접누락 이상
OR NOT    P1060A	// R06 로보트 원위치
AND LOAD
LOAD NOT  K04300	// NG 슈트 개방
OR        P10609	// R06 Arc_On -> PLC
AND LOAD
LOAD NOT  M00050	// 라인 도어열림
OR        P10609	// R06 Arc_On -> PLC
AND LOAD
AND NOT   M10016	// R06 원점 확인 NG
AND NOT   T0055	// 라인1라인 메인에어 압력저하 이상
AND NOT   T0056	// 라인1라인 메인가스 압력저하 이상
LOAD      P10607	// R06 TEACH 모드
LOAD      M0009E	// Line 도어열림
AND       M0009F	// Line 전체 로보트 티칭모드
LOAD NOT  M0009E	// Line 도어열림
AND NOT   M0009F	// Line 전체 로보트 티칭모드
OR LOAD
AND LOAD
OR LOAD
OUT       M1060F	// R06 외부 일시정지
; L17
LOAD      P10607	// R06 TEACH 모드
LOAD      M0009E	// Line 도어열림
AND       M0009F	// Line 전체 로보트 티칭모드
LOAD NOT  M0009E	// Line 도어열림
AND NOT   M0009F	// Line 전체 로보트 티칭모드
OR LOAD
AND LOAD
OUT       M1060D	// R06 외부 티칭모드 신호
; L19
LOAD NOT  M00030	// OP LINE Emergency Stop
AND NOT   M03992	// 절전기동
OUT       M1060E	// R06 외부 비상정지 
; L20
LOAD      F00099
OUT       M10610	// R06 (IN01) 차종1
; L21
LOAD      F0009A
OUT       M10611	// R06 (IN02) 차종2
; L22
LOAD      F0009A
OUT       M10612	// R06 (IN03) 차종3
; L23
LOAD      F0009A
OUT       M10613	// R06 (IN04) 차종4
; L24
LOAD      F0009A
OUT       M10614	// R06 (IN05) 차종5
; L25
LOAD      F0009A
OUT       M10615	// R06 (IN06) 차종6
; L26
LOAD      F0009A
OUT       M10616	// R06 (IN07) 차종7

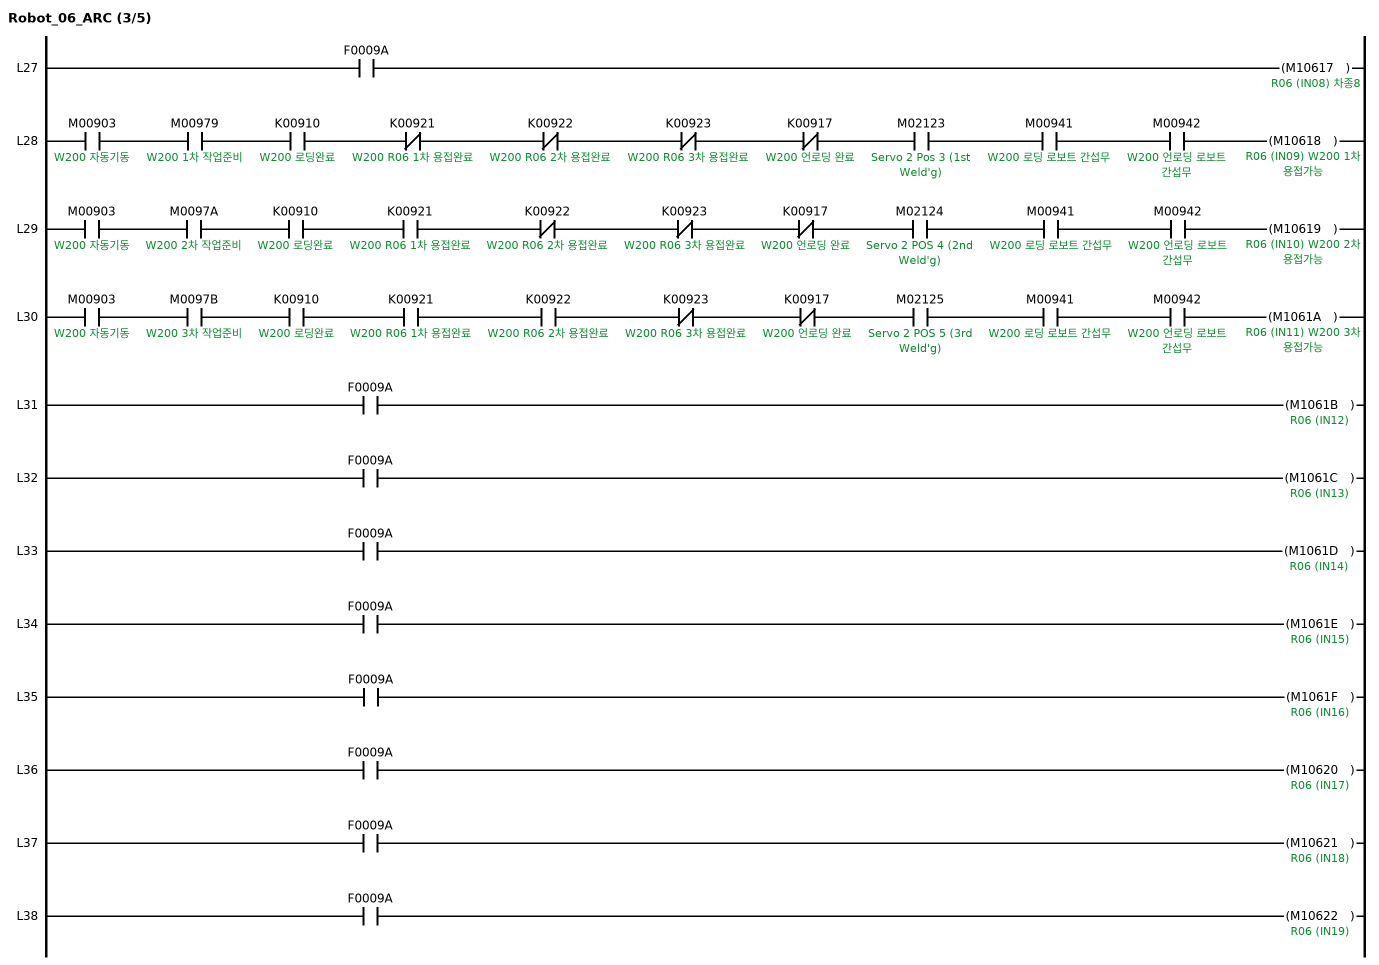
; L27
LOAD      F0009A
OUT       M10617	// R06 (IN08) 차종8
; L28
LOAD      M00903	// W200 자동기동
AND       M00979	// W200 1차 작업준비
AND       K00910	// W200 로딩완료
AND NOT   K00921	// W200 R06 1차 용접완료
AND NOT   K00922	// W200 R06 2차 용접완료
AND NOT   K00923	// W200 R06 3차 용접완료
AND NOT   K00917	// W200 언로딩 완료
AND       M02123	// Servo 2 Pos 3 (1st Weld'g)
AND       M00941	// W200 로딩 로보트 간섭무
AND       M00942	// W200 언로딩 로보트 간섭무
OUT       M10618	// R06 (IN09) W200 1차 용접가능
; L29
LOAD      M00903	// W200 자동기동
AND       M0097A	// W200 2차 작업준비
AND       K00910	// W200 로딩완료
AND       K00921	// W200 R06 1차 용접완료
AND NOT   K00922	// W200 R06 2차 용접완료
AND NOT   K00923	// W200 R06 3차 용접완료
AND NOT   K00917	// W200 언로딩 완료
AND       M02124	// Servo 2 POS 4 (2nd Weld'g)
AND       M00941	// W200 로딩 로보트 간섭무
AND       M00942	// W200 언로딩 로보트 간섭무
OUT       M10619	// R06 (IN10) W200 2차 용접가능
; L30
LOAD      M00903	// W200 자동기동
AND       M0097B	// W200 3차 작업준비
AND       K00910	// W200 로딩완료
AND       K00921	// W200 R06 1차 용접완료
AND       K00922	// W200 R06 2차 용접완료
AND NOT   K00923	// W200 R06 3차 용접완료
AND NOT   K00917	// W200 언로딩 완료
AND       M02125	// Servo 2 POS 5 (3rd Weld'g)
AND       M00941	// W200 로딩 로보트 간섭무
AND       M00942	// W200 언로딩 로보트 간섭무
OUT       M1061A	// R06 (IN11) W200 3차 용접가능
; L31
LOAD      F0009A
OUT       M1061B	// R06 (IN12)
; L32
LOAD      F0009A
OUT       M1061C	// R06 (IN13)
; L33
LOAD      F0009A
OUT       M1061D	// R06 (IN14)
; L34
LOAD      F0009A
OUT       M1061E	// R06 (IN15)
; L35
LOAD      F0009A
OUT       M1061F	// R06 (IN16)
; L36
LOAD      F0009A
OUT       M10620	// R06 (IN17)
; L37
LOAD      F0009A
OUT       M10621	// R06 (IN18)
; L38
LOAD      F0009A
OUT       M10622	// R06 (IN19)

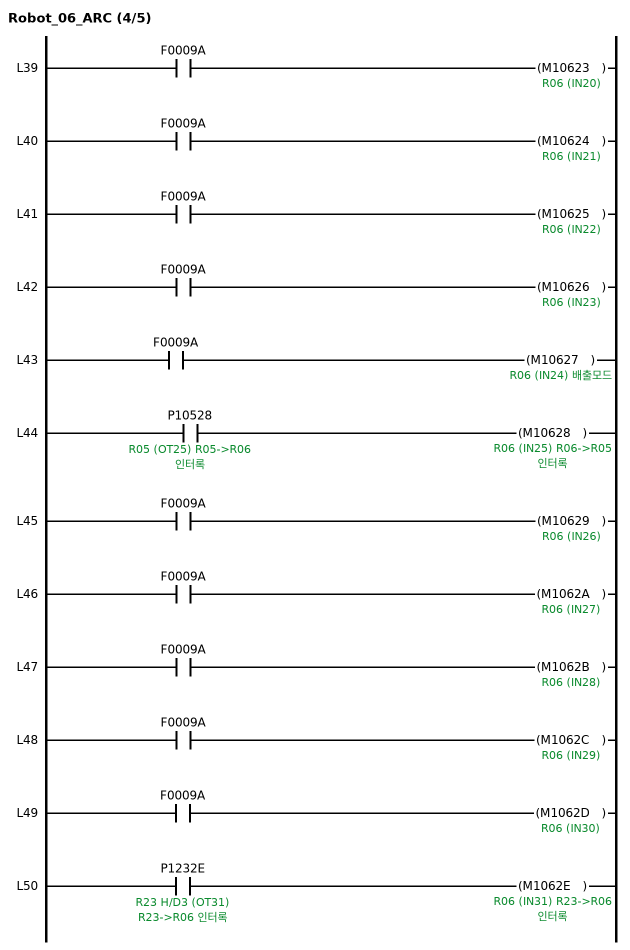
; L39
LOAD      F0009A
OUT       M10623	// R06 (IN20)
; L40
LOAD      F0009A
OUT       M10624	// R06 (IN21)
; L41
LOAD      F0009A
OUT       M10625	// R06 (IN22)
; L42
LOAD      F0009A
OUT       M10626	// R06 (IN23)
; L43
LOAD      F0009A
OUT       M10627	// R06 (IN24) 배출모드
; L44
LOAD      P10528	// R05 (OT25) R05->R06 인터록
OUT       M10628	// R06 (IN25) R06->R05 인터록
; L45
LOAD      F0009A
OUT       M10629	// R06 (IN26)
; L46
LOAD      F0009A
OUT       M1062A	// R06 (IN27)
; L47
LOAD      F0009A
OUT       M1062B	// R06 (IN28)
; L48
LOAD      F0009A
OUT       M1062C	// R06 (IN29)
; L49
LOAD      F0009A
OUT       M1062D	// R06 (IN30)
; L50
LOAD      P1232E	// R23 H/D3 (OT31) R23->R06 인터록
OUT       M1062E	// R06 (IN31) R23->R06 인터록

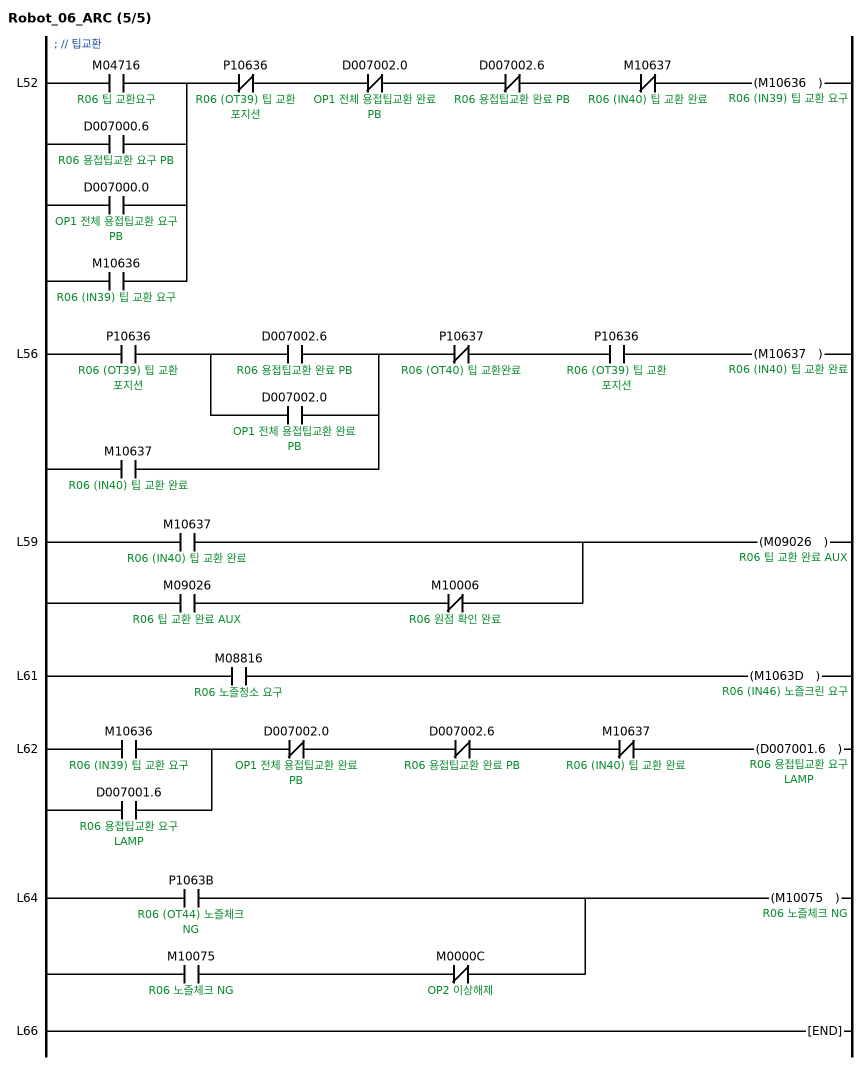
//  // 팁교환
; L52
LOAD      M04716	// R06 팁 교환요구
OR        D007000.6	// R06 용접팁교환 요구 PB
OR        D007000.0	// OP1 전체 용접팁교환 요구 PB
OR        M10636	// R06 (IN39) 팁 교환 요구
AND NOT   P10636	// R06 (OT39) 팁 교환 포지션
AND NOT   D007002.0	// OP1 전체 용접팁교환 완료 PB
AND NOT   D007002.6	// R06 용접팁교환 완료 PB
AND NOT   M10637	// R06 (IN40) 팁 교환 완료
OUT       M10636	// R06 (IN39) 팁 교환 요구
; L56
LOAD      P10636	// R06 (OT39) 팁 교환 포지션
LOAD      D007002.6	// R06 용접팁교환 완료 PB
OR        D007002.0	// OP1 전체 용접팁교환 완료 PB
AND LOAD
OR        M10637	// R06 (IN40) 팁 교환 완료
AND NOT   P10637	// R06 (OT40) 팁 교환완료
AND       P10636	// R06 (OT39) 팁 교환 포지션
OUT       M10637	// R06 (IN40) 팁 교환 완료
; L59
LOAD      M10637	// R06 (IN40) 팁 교환 완료
LOAD      M09026	// R06 팁 교환 완료 AUX
AND NOT   M10006	// R06 원점 확인 완료
OR LOAD
OUT       M09026	// R06 팁 교환 완료 AUX
; L61
LOAD      M08816	// R06 노즐청소 요구
OUT       M1063D	// R06 (IN46) 노즐크린 요구
; L62
LOAD      M10636	// R06 (IN39) 팁 교환 요구
OR        D007001.6	// R06 용접팁교환 요구 LAMP
AND NOT   D007002.0	// OP1 전체 용접팁교환 완료 PB
AND NOT   D007002.6	// R06 용접팁교환 완료 PB
AND NOT   M10637	// R06 (IN40) 팁 교환 완료
OUT       D007001.6	// R06 용접팁교환 요구 LAMP
; L64
LOAD      P1063B	// R06 (OT44) 노즐체크 NG
LOAD      M10075	// R06 노즐체크 NG
AND NOT   M0000C	// OP2 이상해제
OR LOAD
OUT       M10075	// R06 노즐체크 NG
; L66
END

PROGRAM Robot_21_HD1 (task: 스캔 프로그램)

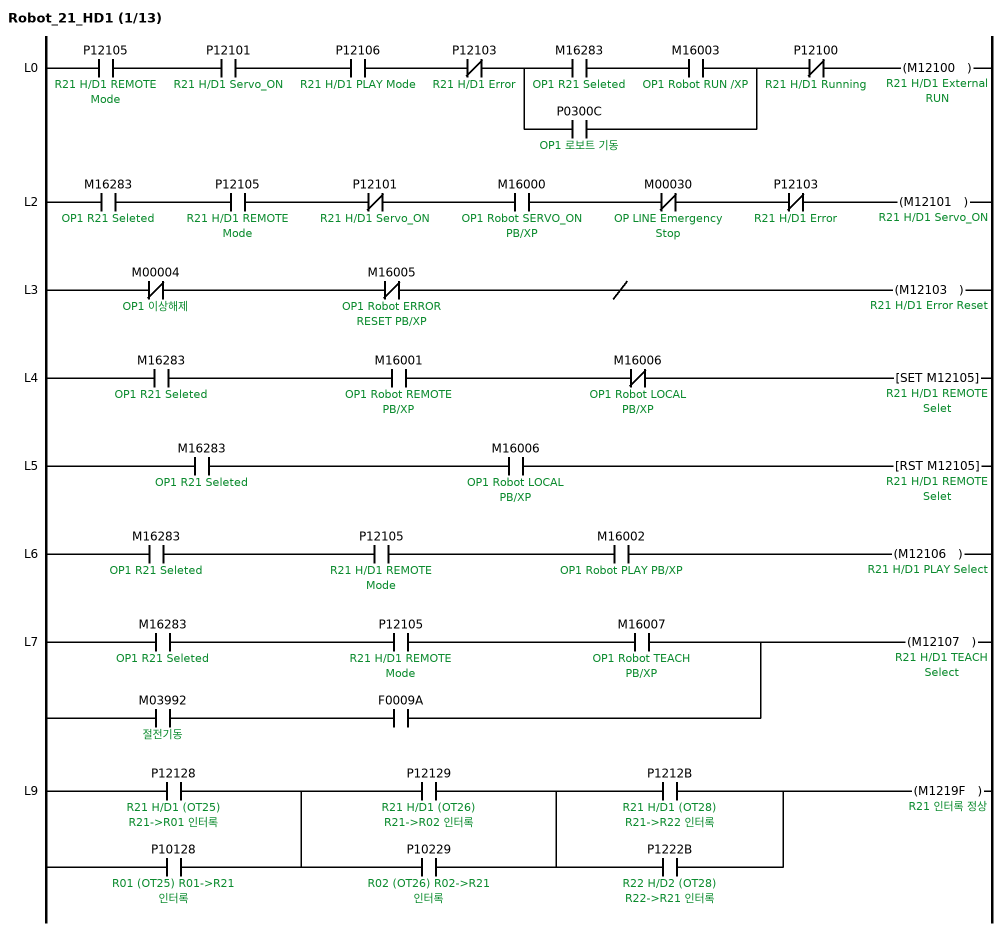
; L0
LOAD      P12105	// R21 H/D1 REMOTE Mode
AND       P12101	// R21 H/D1 Servo_ON
AND       P12106	// R21 H/D1 PLAY Mode
AND NOT   P12103	// R21 H/D1 Error
LOAD      M16283	// OP1 R21 Seleted
AND       M16003	// OP1 Robot RUN /XP
OR        P0300C	// OP1 로보트 기동
AND LOAD
AND NOT   P12100	// R21 H/D1 Running
OUT       M12100	// R21 H/D1 External RUN
; L2
LOAD      M16283	// OP1 R21 Seleted
AND       P12105	// R21 H/D1 REMOTE Mode
AND NOT   P12101	// R21 H/D1 Servo_ON
AND       M16000	// OP1 Robot SERVO_ON PB/XP
AND NOT   M00030	// OP LINE Emergency Stop
AND NOT   P12103	// R21 H/D1 Error
OUT       M12101	// R21 H/D1 Servo_ON
; L3
LOAD NOT  M00004	// OP1 이상해제
AND NOT   M16005	// OP1 Robot ERROR RESET PB/XP
NOT
OUT       M12103	// R21 H/D1 Error Reset
; L4
LOAD      M16283	// OP1 R21 Seleted
AND       M16001	// OP1 Robot REMOTE PB/XP
AND NOT   M16006	// OP1 Robot LOCAL PB/XP
SET       M12105	// R21 H/D1 REMOTE Selet
; L5
LOAD      M16283	// OP1 R21 Seleted
AND       M16006	// OP1 Robot LOCAL PB/XP
RST       M12105	// R21 H/D1 REMOTE Selet
; L6
LOAD      M16283	// OP1 R21 Seleted
AND       P12105	// R21 H/D1 REMOTE Mode
AND       M16002	// OP1 Robot PLAY PB/XP
OUT       M12106	// R21 H/D1 PLAY Select
; L7
LOAD      M16283	// OP1 R21 Seleted
AND       P12105	// R21 H/D1 REMOTE Mode
AND       M16007	// OP1 Robot TEACH PB/XP
LOAD      M03992	// 절전기동
AND       F0009A
OR LOAD
OUT       M12107	// R21 H/D1 TEACH Select
; L9
LOAD      P12128	// R21 H/D1 (OT25) R21->R01 인터록
OR        P10128	// R01 (OT25) R01->R21 인터록
LOAD      P12129	// R21 H/D1 (OT26) R21->R02 인터록
OR        P10229	// R02 (OT26) R02->R21 인터록
AND LOAD
LOAD      P1212B	// R21 H/D1 (OT28) R21->R22 인터록
OR        P1222B	// R22 H/D2 (OT28) R22->R21 인터록
AND LOAD
OUT       M1219F	// R21 인터록 정상

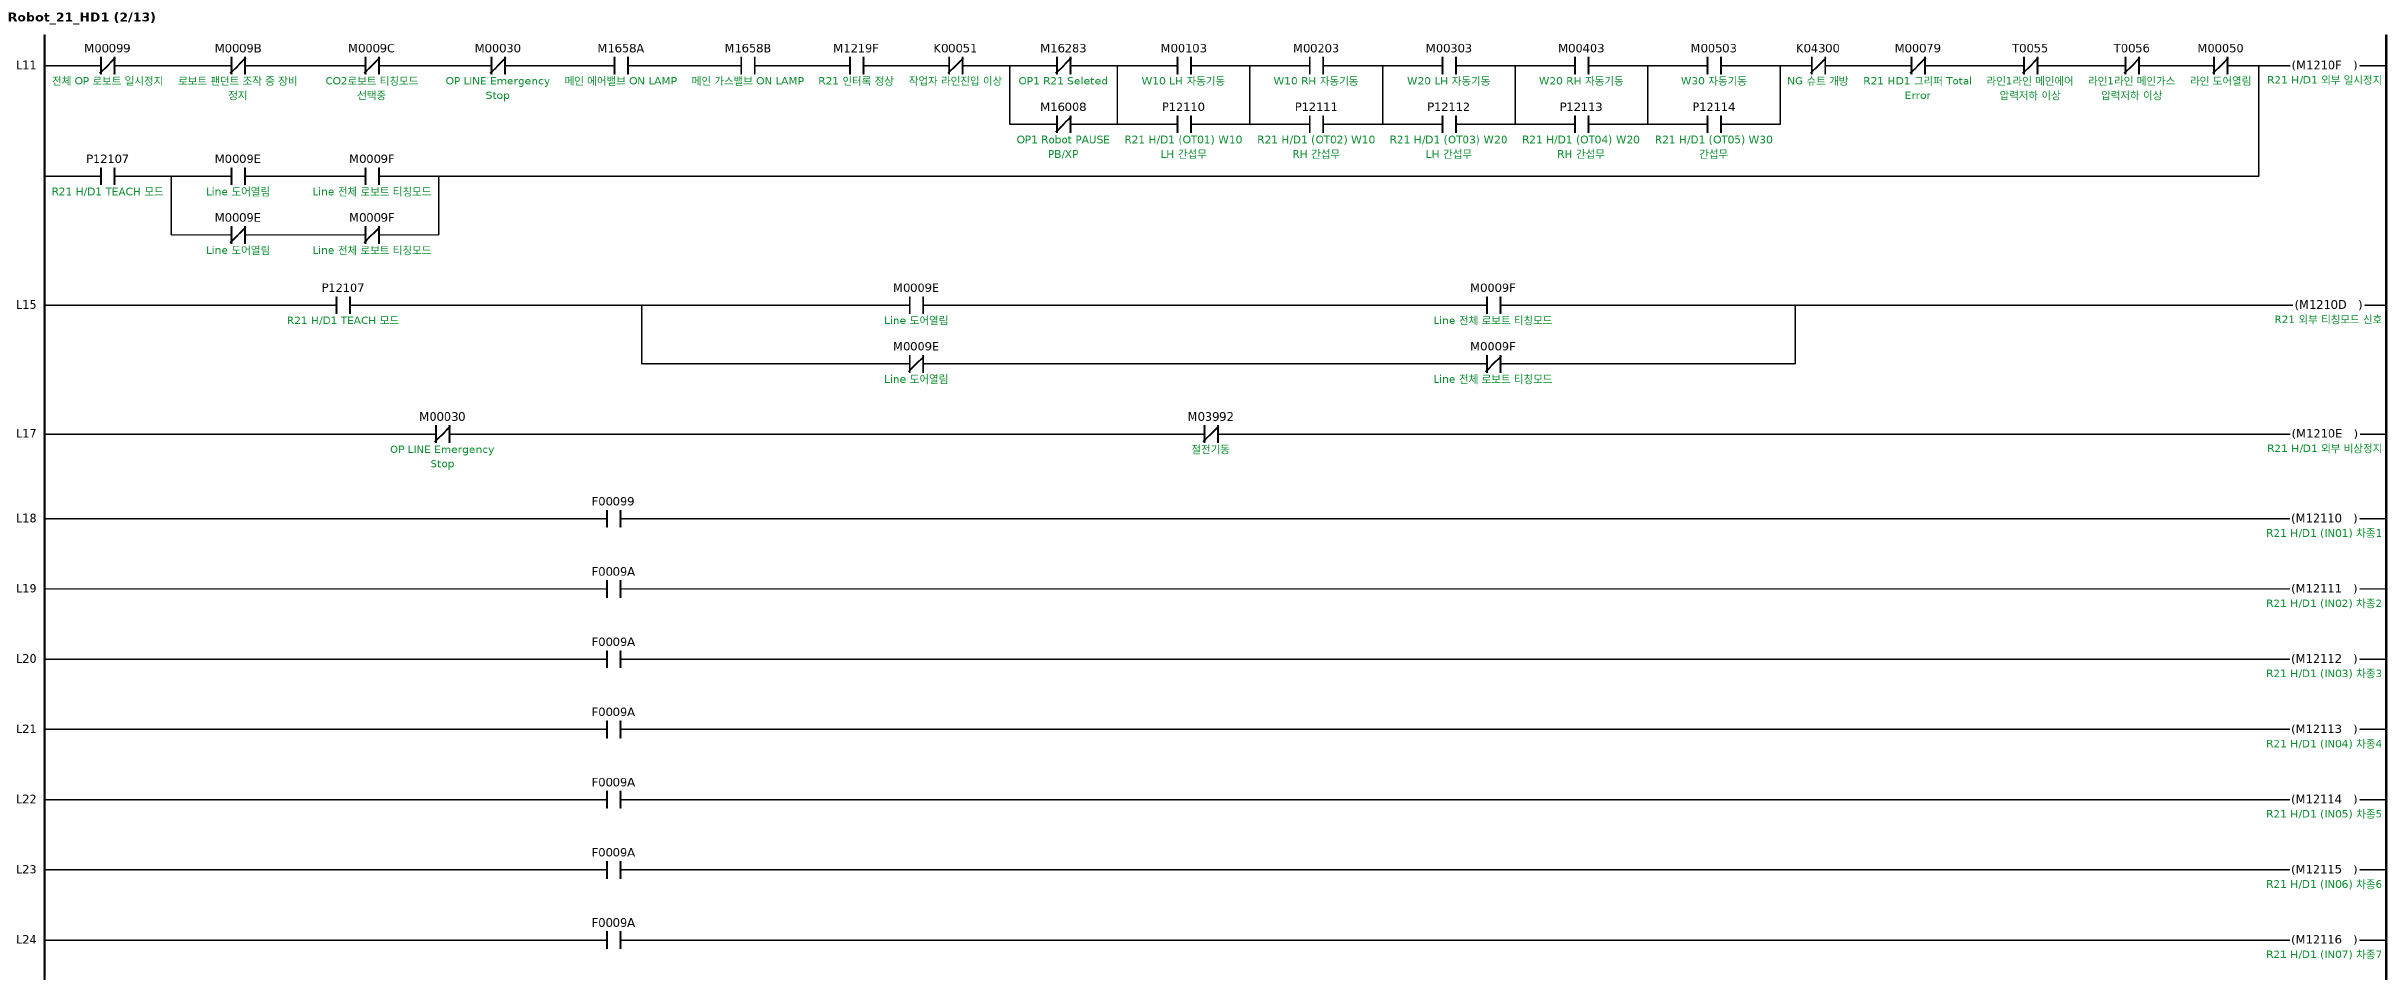
; L11
LOAD NOT  M00099	// 전체 OP 로보트 일시정지
AND NOT   M0009B	// 로보트 팬던트 조작 중 장비 정지
AND NOT   M0009C	// CO2로보트 티칭모드 선택중
AND NOT   M00030	// OP LINE Emergency Stop
AND       M1658A	// 메인 에어밸브 ON LAMP
AND       M1658B	// 메인 가스밸브 ON LAMP
AND       M1219F	// R21 인터록 정상
AND NOT   K00051	//  작업자 라인진입 이상
LOAD NOT  M16283	// OP1 R21 Seleted
OR NOT    M16008	// OP1 Robot PAUSE PB/XP
AND LOAD
LOAD      M00103	// W10 LH 자동기동
OR        P12110	// R21 H/D1 (OT01) W10 LH 간섭무
AND LOAD
LOAD      M00203	// W10 RH 자동기동
OR        P12111	// R21 H/D1 (OT02) W10 RH 간섭무
AND LOAD
LOAD      M00303	// W20 LH 자동기동
OR        P12112	// R21 H/D1 (OT03) W20 LH 간섭무
AND LOAD
LOAD      M00403	// W20 RH 자동기동
OR        P12113	// R21 H/D1 (OT04) W20 RH 간섭무
AND LOAD
LOAD      M00503	// W30 자동기동
OR        P12114	// R21 H/D1 (OT05) W30 간섭무
AND LOAD
AND NOT   K04300	// NG 슈트 개방
AND NOT   M00079	// R21 HD1 그리퍼 Total Error 
AND NOT   T0055	// 라인1라인 메인에어 압력저하 이상
AND NOT   T0056	// 라인1라인 메인가스 압력저하 이상
AND NOT   M00050	// 라인 도어열림
LOAD      P12107	// R21 H/D1 TEACH 모드
LOAD      M0009E	// Line 도어열림
AND       M0009F	// Line 전체 로보트 티칭모드
LOAD NOT  M0009E	// Line 도어열림
AND NOT   M0009F	// Line 전체 로보트 티칭모드
OR LOAD
AND LOAD
OR LOAD
OUT       M1210F	// R21 H/D1 외부 일시정지
; L15
LOAD      P12107	// R21 H/D1 TEACH 모드
LOAD      M0009E	// Line 도어열림
AND       M0009F	// Line 전체 로보트 티칭모드
LOAD NOT  M0009E	// Line 도어열림
AND NOT   M0009F	// Line 전체 로보트 티칭모드
OR LOAD
AND LOAD
OUT       M1210D	// R21 외부 티칭모드 신호
; L17
LOAD NOT  M00030	// OP LINE Emergency Stop
AND NOT   M03992	// 절전기동
OUT       M1210E	// R21 H/D1 외부 비상정지 
; L18
LOAD      F00099
OUT       M12110	// R21 H/D1 (IN01) 차종1
; L19
LOAD      F0009A
OUT       M12111	// R21 H/D1 (IN02) 차종2
; L20
LOAD      F0009A
OUT       M12112	// R21 H/D1 (IN03) 차종3
; L21
LOAD      F0009A
OUT       M12113	// R21 H/D1 (IN04) 차종4
; L22
LOAD      F0009A
OUT       M12114	// R21 H/D1 (IN05) 차종5
; L23
LOAD      F0009A
OUT       M12115	// R21 H/D1 (IN06) 차종6
; L24
LOAD      F0009A
OUT       M12116	// R21 H/D1 (IN07) 차종7

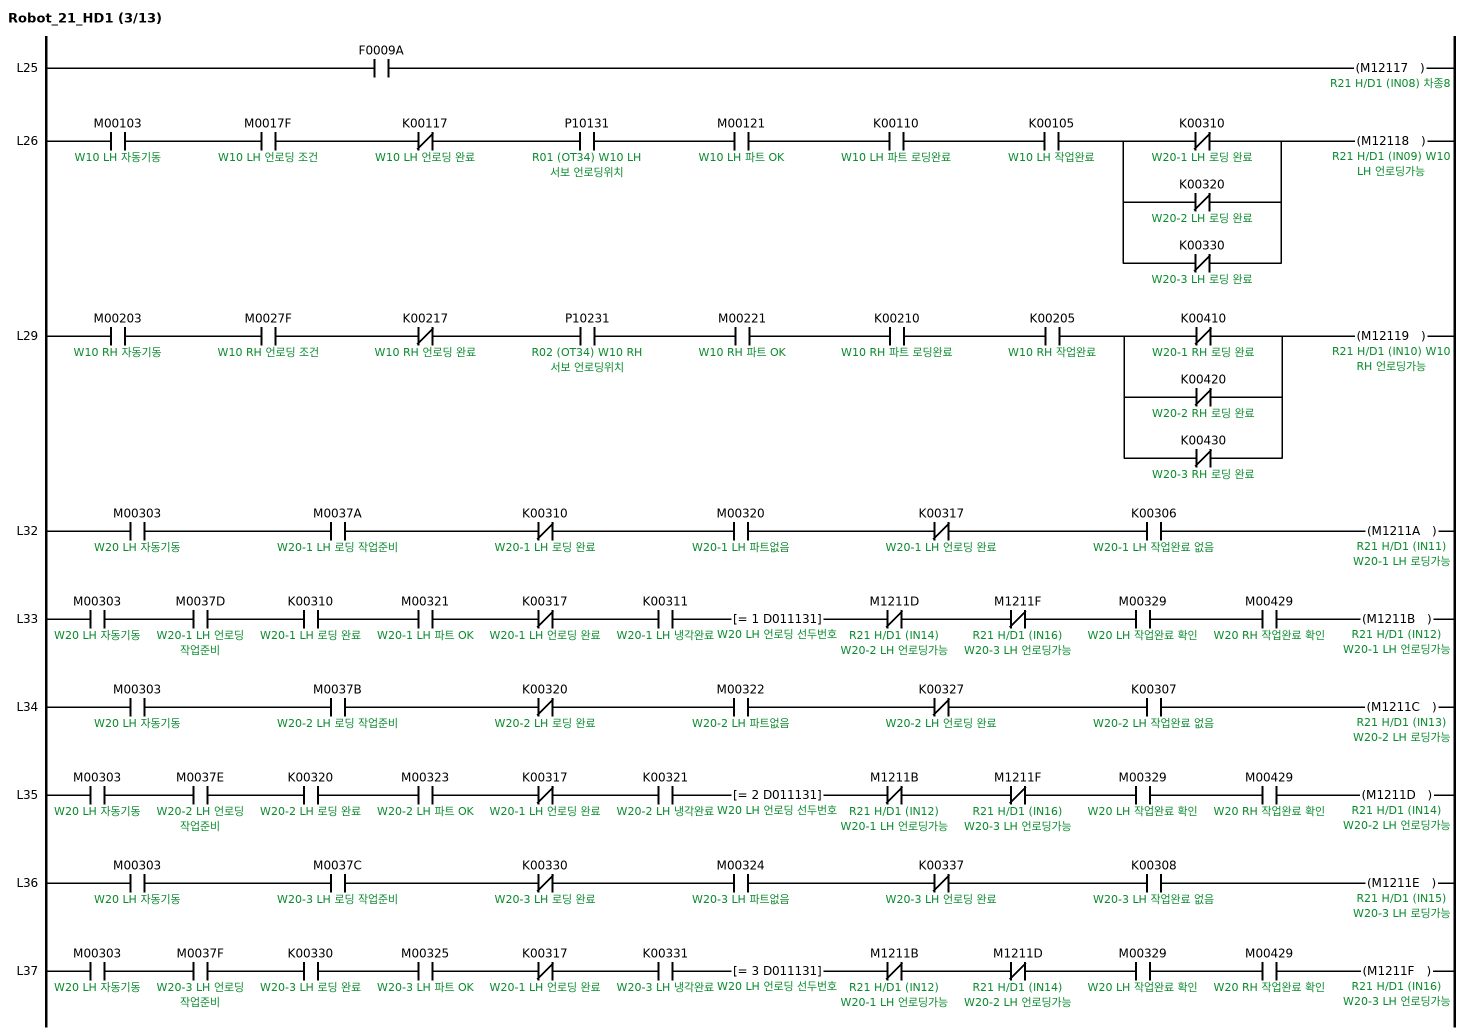
; L25
LOAD      F0009A
OUT       M12117	// R21 H/D1 (IN08) 차종8
; L26
LOAD      M00103	// W10 LH 자동기동
AND       M0017F	// W10 LH 언로딩 조건
AND NOT   K00117	// W10 LH 언로딩 완료
AND       P10131	// R01 (OT34) W10 LH 서보 언로딩위치
AND       M00121	// W10 LH 파트 OK
AND       K00110	// W10 LH 파트 로딩완료
AND       K00105	// W10 LH 작업완료
LOAD NOT  K00310	// W20-1 LH 로딩 완료
OR NOT    K00320	// W20-2 LH 로딩 완료
OR NOT    K00330	// W20-3 LH 로딩 완료
AND LOAD
OUT       M12118	// R21 H/D1 (IN09) W10 LH 언로딩가능
; L29
LOAD      M00203	// W10 RH 자동기동
AND       M0027F	// W10 RH 언로딩 조건
AND NOT   K00217	// W10 RH 언로딩 완료
AND       P10231	// R02 (OT34) W10 RH 서보 언로딩위치
AND       M00221	// W10 RH 파트 OK
AND       K00210	// W10 RH 파트 로딩완료
AND       K00205	// W10 RH 작업완료
LOAD NOT  K00410	// W20-1 RH 로딩 완료
OR NOT    K00420	// W20-2 RH 로딩 완료
OR NOT    K00430	// W20-3 RH 로딩 완료
AND LOAD
OUT       M12119	// R21 H/D1 (IN10) W10 RH 언로딩가능
; L32
LOAD      M00303	// W20 LH 자동기동
AND       M0037A	// W20-1 LH 로딩 작업준비
AND NOT   K00310	// W20-1 LH 로딩 완료
AND       M00320	// W20-1 LH 파트없음
AND NOT   K00317	// W20-1 LH 언로딩 완료
AND       K00306	// W20-1 LH 작업완료 없음
OUT       M1211A	// R21 H/D1 (IN11) W20-1 LH 로딩가능
; L33
LOAD      M00303	// W20 LH 자동기동
AND       M0037D	// W20-1 LH 언로딩 작업준비
AND       K00310	// W20-1 LH 로딩 완료
AND       M00321	// W20-1 LH 파트 OK
AND NOT   K00317	// W20-1 LH 언로딩 완료
AND       K00311	// W20-1 LH 냉각완료
AND=      1 D011131	// W20 LH 언로딩 선두번호
AND NOT   M1211D	// R21 H/D1 (IN14) W20-2 LH 언로딩가능
AND NOT   M1211F	// R21 H/D1 (IN16) W20-3 LH 언로딩가능
AND       M00329	// W20 LH 작업완료 확인
AND       M00429	// W20 RH 작업완료 확인
OUT       M1211B	// R21 H/D1 (IN12) W20-1 LH 언로딩가능
; L34
LOAD      M00303	// W20 LH 자동기동
AND       M0037B	// W20-2 LH 로딩 작업준비
AND NOT   K00320	// W20-2 LH 로딩 완료
AND       M00322	// W20-2 LH 파트없음
AND NOT   K00327	// W20-2 LH 언로딩 완료
AND       K00307	// W20-2 LH 작업완료 없음
OUT       M1211C	// R21 H/D1 (IN13) W20-2 LH 로딩가능
; L35
LOAD      M00303	// W20 LH 자동기동
AND       M0037E	// W20-2 LH 언로딩 작업준비
AND       K00320	// W20-2 LH 로딩 완료
AND       M00323	// W20-2 LH 파트 OK
AND NOT   K00317	// W20-1 LH 언로딩 완료
AND       K00321	// W20-2 LH 냉각완료
AND=      2 D011131	// W20 LH 언로딩 선두번호
AND NOT   M1211B	// R21 H/D1 (IN12) W20-1 LH 언로딩가능
AND NOT   M1211F	// R21 H/D1 (IN16) W20-3 LH 언로딩가능
AND       M00329	// W20 LH 작업완료 확인
AND       M00429	// W20 RH 작업완료 확인
OUT       M1211D	// R21 H/D1 (IN14) W20-2 LH 언로딩가능
; L36
LOAD      M00303	// W20 LH 자동기동
AND       M0037C	// W20-3 LH 로딩 작업준비
AND NOT   K00330	// W20-3 LH 로딩 완료
AND       M00324	// W20-3 LH 파트없음
AND NOT   K00337	// W20-3 LH 언로딩 완료
AND       K00308	// W20-3 LH 작업완료 없음
OUT       M1211E	// R21 H/D1 (IN15) W20-3 LH 로딩가능
; L37
LOAD      M00303	// W20 LH 자동기동
AND       M0037F	// W20-3 LH 언로딩 작업준비
AND       K00330	// W20-3 LH 로딩 완료
AND       M00325	// W20-3 LH 파트 OK
AND NOT   K00317	// W20-1 LH 언로딩 완료
AND       K00331	// W20-3 LH 냉각완료
AND=      3 D011131	// W20 LH 언로딩 선두번호
AND NOT   M1211B	// R21 H/D1 (IN12) W20-1 LH 언로딩가능
AND NOT   M1211D	// R21 H/D1 (IN14) W20-2 LH 언로딩가능
AND       M00329	// W20 LH 작업완료 확인
AND       M00429	// W20 RH 작업완료 확인
OUT       M1211F	// R21 H/D1 (IN16) W20-3 LH 언로딩가능

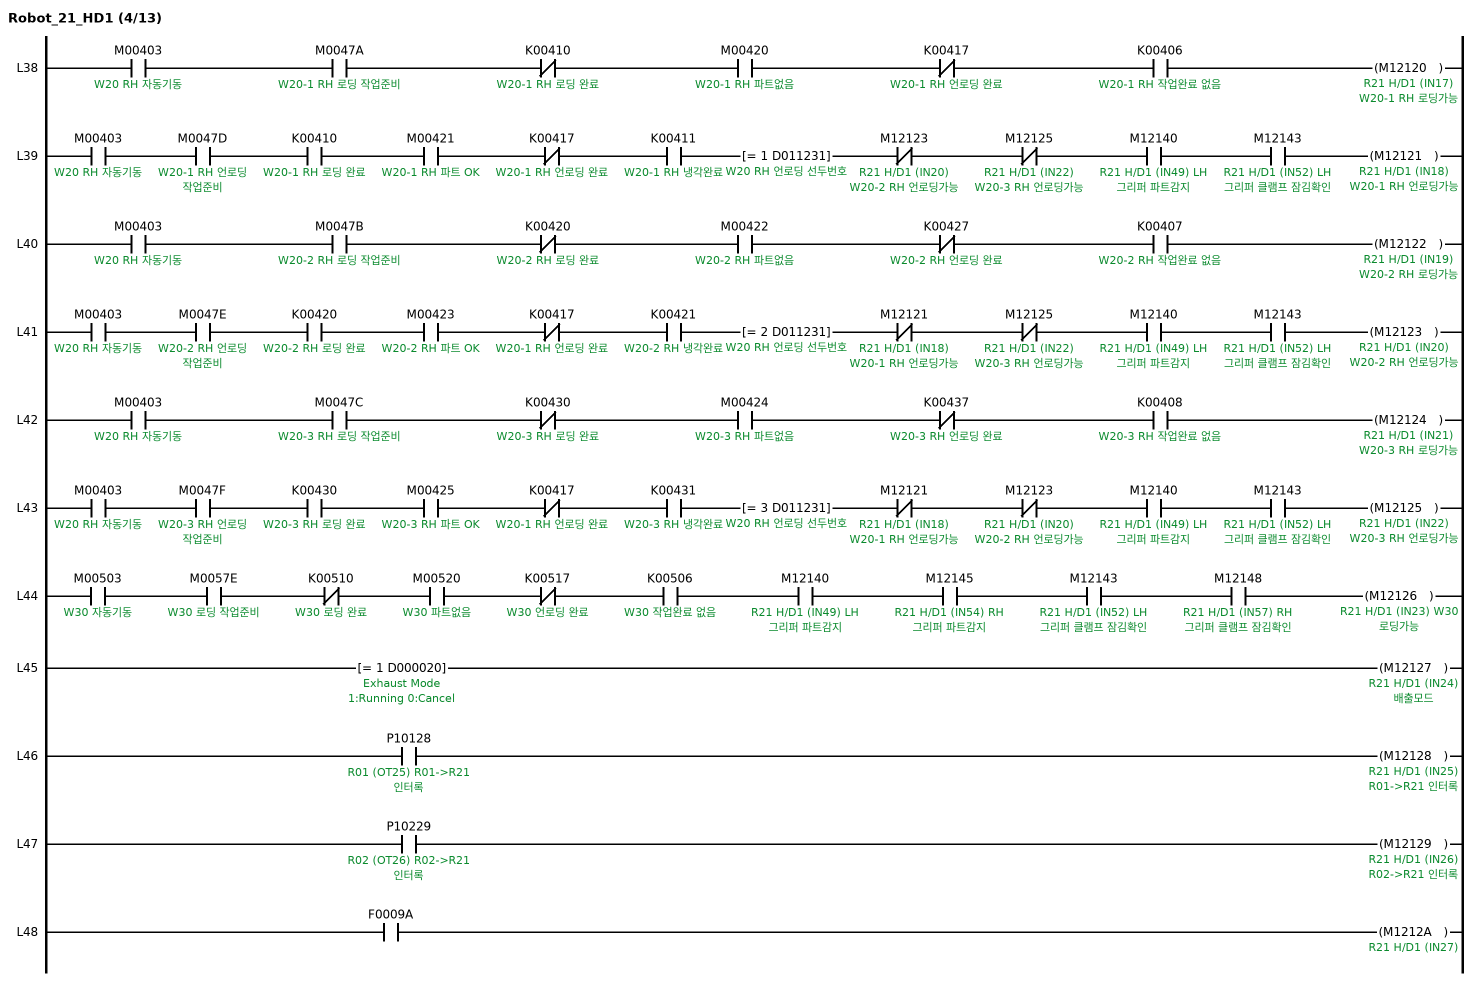
; L38
LOAD      M00403	// W20 RH 자동기동
AND       M0047A	// W20-1 RH 로딩 작업준비
AND NOT   K00410	// W20-1 RH 로딩 완료
AND       M00420	// W20-1 RH 파트없음
AND NOT   K00417	// W20-1 RH 언로딩 완료
AND       K00406	// W20-1 RH 작업완료 없음
OUT       M12120	// R21 H/D1 (IN17) W20-1 RH 로딩가능
; L39
LOAD      M00403	// W20 RH 자동기동
AND       M0047D	// W20-1 RH 언로딩 작업준비
AND       K00410	// W20-1 RH 로딩 완료
AND       M00421	// W20-1 RH 파트 OK
AND NOT   K00417	// W20-1 RH 언로딩 완료
AND       K00411	// W20-1 RH 냉각완료
AND=      1 D011231	// W20 RH 언로딩 선두번호
AND NOT   M12123	// R21 H/D1 (IN20) W20-2 RH 언로딩가능
AND NOT   M12125	// R21 H/D1 (IN22) W20-3 RH 언로딩가능
AND       M12140	// R21 H/D1 (IN49) LH 그리퍼 파트감지
AND       M12143	// R21 H/D1 (IN52) LH 그리퍼 클램프 잠김확인
OUT       M12121	// R21 H/D1 (IN18) W20-1 RH 언로딩가능
; L40
LOAD      M00403	// W20 RH 자동기동
AND       M0047B	// W20-2 RH 로딩 작업준비
AND NOT   K00420	// W20-2 RH 로딩 완료
AND       M00422	// W20-2 RH 파트없음
AND NOT   K00427	// W20-2 RH 언로딩 완료
AND       K00407	// W20-2 RH 작업완료 없음
OUT       M12122	// R21 H/D1 (IN19) W20-2 RH 로딩가능
; L41
LOAD      M00403	// W20 RH 자동기동
AND       M0047E	// W20-2 RH 언로딩 작업준비
AND       K00420	// W20-2 RH 로딩 완료
AND       M00423	// W20-2 RH 파트 OK
AND NOT   K00417	// W20-1 RH 언로딩 완료
AND       K00421	// W20-2 RH 냉각완료
AND=      2 D011231	// W20 RH 언로딩 선두번호
AND NOT   M12121	// R21 H/D1 (IN18) W20-1 RH 언로딩가능
AND NOT   M12125	// R21 H/D1 (IN22) W20-3 RH 언로딩가능
AND       M12140	// R21 H/D1 (IN49) LH 그리퍼 파트감지
AND       M12143	// R21 H/D1 (IN52) LH 그리퍼 클램프 잠김확인
OUT       M12123	// R21 H/D1 (IN20) W20-2 RH 언로딩가능
; L42
LOAD      M00403	// W20 RH 자동기동
AND       M0047C	// W20-3 RH 로딩 작업준비
AND NOT   K00430	// W20-3 RH 로딩 완료
AND       M00424	// W20-3 RH 파트없음
AND NOT   K00437	// W20-3 RH 언로딩 완료
AND       K00408	// W20-3 RH 작업완료 없음
OUT       M12124	// R21 H/D1 (IN21) W20-3 RH 로딩가능
; L43
LOAD      M00403	// W20 RH 자동기동
AND       M0047F	// W20-3 RH 언로딩 작업준비
AND       K00430	// W20-3 RH 로딩 완료
AND       M00425	// W20-3 RH 파트 OK
AND NOT   K00417	// W20-1 RH 언로딩 완료
AND       K00431	// W20-3 RH 냉각완료
AND=      3 D011231	// W20 RH 언로딩 선두번호
AND NOT   M12121	// R21 H/D1 (IN18) W20-1 RH 언로딩가능
AND NOT   M12123	// R21 H/D1 (IN20) W20-2 RH 언로딩가능
AND       M12140	// R21 H/D1 (IN49) LH 그리퍼 파트감지
AND       M12143	// R21 H/D1 (IN52) LH 그리퍼 클램프 잠김확인
OUT       M12125	// R21 H/D1 (IN22) W20-3 RH 언로딩가능
; L44
LOAD      M00503	// W30 자동기동
AND       M0057E	// W30 로딩 작업준비
AND NOT   K00510	// W30 로딩 완료
AND       M00520	// W30 파트없음
AND NOT   K00517	// W30 언로딩 완료
AND       K00506	// W30 작업완료 없음
AND       M12140	// R21 H/D1 (IN49) LH 그리퍼 파트감지
AND       M12145	// R21 H/D1 (IN54) RH 그리퍼 파트감지
AND       M12143	// R21 H/D1 (IN52) LH 그리퍼 클램프 잠김확인
AND       M12148	// R21 H/D1 (IN57) RH 그리퍼 클램프 잠김확인
OUT       M12126	// R21 H/D1 (IN23) W30 로딩가능
; L45
LOAD=     1 D000020	// Exhaust Mode 1:Running 0:Cancel
OUT       M12127	// R21 H/D1 (IN24) 배출모드
; L46
LOAD      P10128	// R01 (OT25) R01->R21 인터록
OUT       M12128	// R21 H/D1 (IN25) R01->R21 인터록
; L47
LOAD      P10229	// R02 (OT26) R02->R21 인터록
OUT       M12129	// R21 H/D1 (IN26) R02->R21 인터록
; L48
LOAD      F0009A
OUT       M1212A	// R21 H/D1 (IN27)

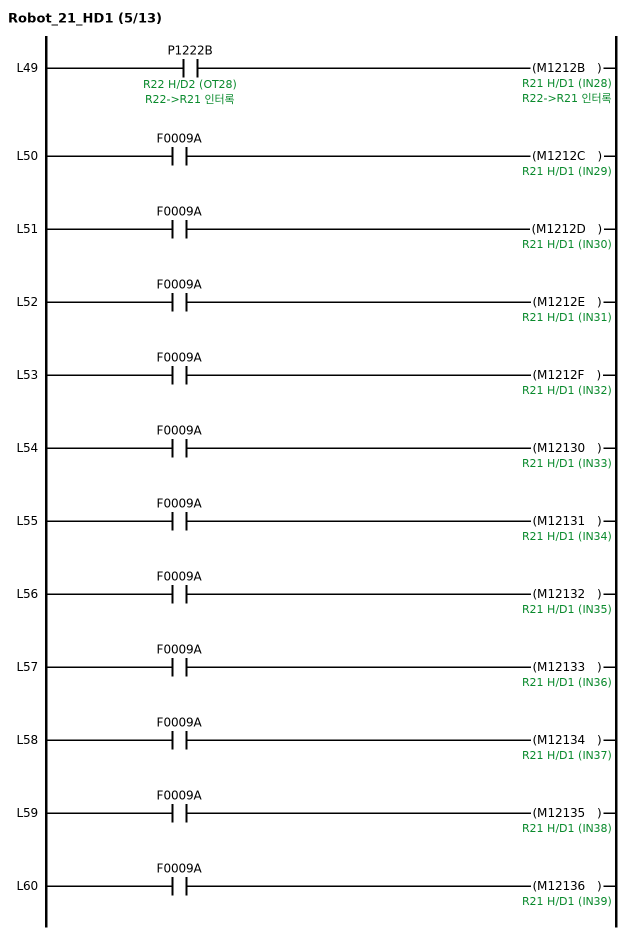
; L49
LOAD      P1222B	// R22 H/D2 (OT28) R22->R21 인터록
OUT       M1212B	// R21 H/D1 (IN28) R22->R21 인터록
; L50
LOAD      F0009A
OUT       M1212C	// R21 H/D1 (IN29)
; L51
LOAD      F0009A
OUT       M1212D	// R21 H/D1 (IN30)
; L52
LOAD      F0009A
OUT       M1212E	// R21 H/D1 (IN31)
; L53
LOAD      F0009A
OUT       M1212F	// R21 H/D1 (IN32)
; L54
LOAD      F0009A
OUT       M12130	// R21 H/D1 (IN33)
; L55
LOAD      F0009A
OUT       M12131	// R21 H/D1 (IN34)
; L56
LOAD      F0009A
OUT       M12132	// R21 H/D1 (IN35)
; L57
LOAD      F0009A
OUT       M12133	// R21 H/D1 (IN36)
; L58
LOAD      F0009A
OUT       M12134	// R21 H/D1 (IN37)
; L59
LOAD      F0009A
OUT       M12135	// R21 H/D1 (IN38)
; L60
LOAD      F0009A
OUT       M12136	// R21 H/D1 (IN39)

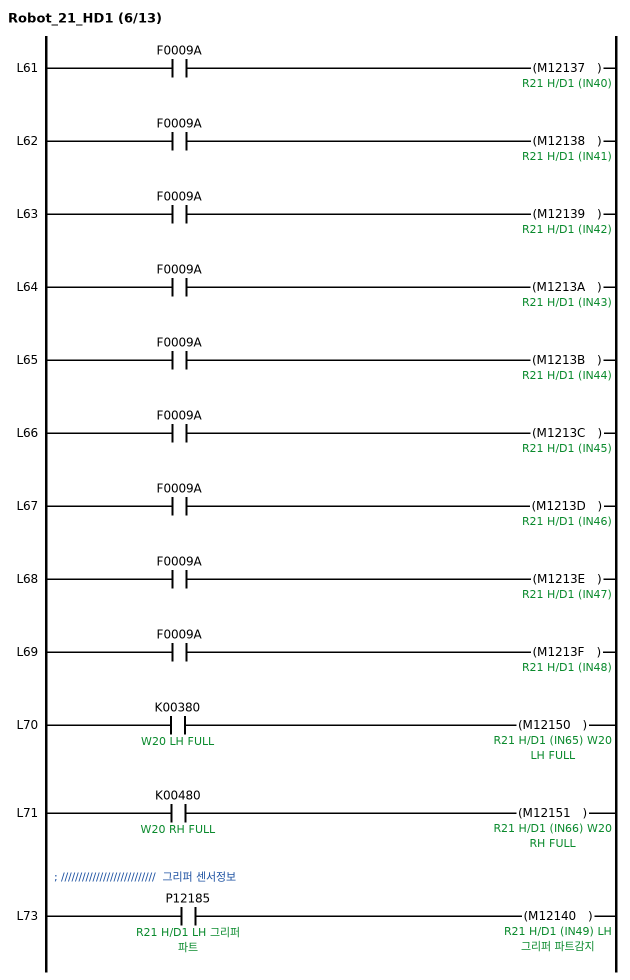
; L61
LOAD      F0009A
OUT       M12137	// R21 H/D1 (IN40)
; L62
LOAD      F0009A
OUT       M12138	// R21 H/D1 (IN41)
; L63
LOAD      F0009A
OUT       M12139	// R21 H/D1 (IN42)
; L64
LOAD      F0009A
OUT       M1213A	// R21 H/D1 (IN43)
; L65
LOAD      F0009A
OUT       M1213B	// R21 H/D1 (IN44)
; L66
LOAD      F0009A
OUT       M1213C	// R21 H/D1 (IN45)
; L67
LOAD      F0009A
OUT       M1213D	// R21 H/D1 (IN46)
; L68
LOAD      F0009A
OUT       M1213E	// R21 H/D1 (IN47)
; L69
LOAD      F0009A
OUT       M1213F	// R21 H/D1 (IN48)
; L70
LOAD      K00380	// W20 LH FULL
OUT       M12150	// R21 H/D1 (IN65) W20 LH FULL
; L71
LOAD      K00480	// W20 RH FULL
OUT       M12151	// R21 H/D1 (IN66) W20 RH FULL
// ///////////////////////////  그리퍼 센서정보
; L73
LOAD      P12185	// R21 H/D1 LH 그리퍼 파트
OUT       M12140	// R21 H/D1 (IN49) LH 그리퍼 파트감지

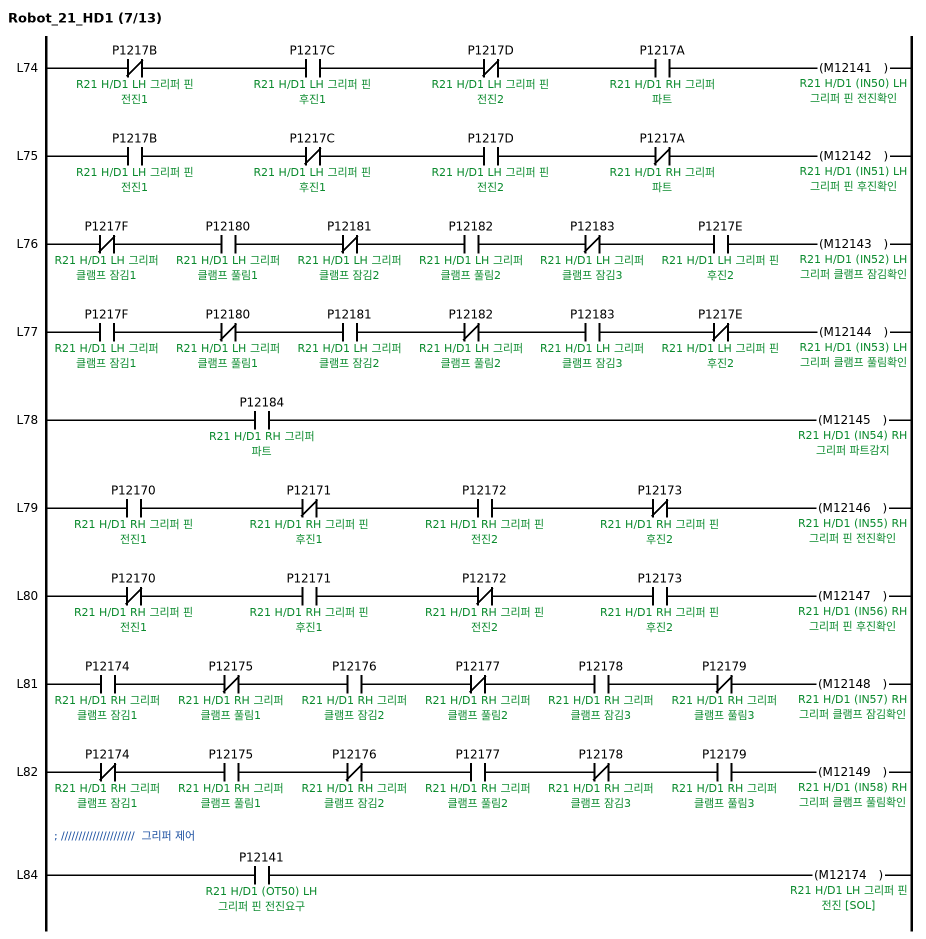
; L74
LOAD NOT  P1217B	// R21 H/D1 LH 그리퍼 핀 전진1
AND       P1217C	// R21 H/D1 LH 그리퍼 핀 후진1
AND NOT   P1217D	// R21 H/D1 LH 그리퍼 핀 전진2
AND       P1217A	// R21 H/D1 RH 그리퍼 파트
OUT       M12141	// R21 H/D1 (IN50) LH 그리퍼 핀 전진확인
; L75
LOAD      P1217B	// R21 H/D1 LH 그리퍼 핀 전진1
AND NOT   P1217C	// R21 H/D1 LH 그리퍼 핀 후진1
AND       P1217D	// R21 H/D1 LH 그리퍼 핀 전진2
AND NOT   P1217A	// R21 H/D1 RH 그리퍼 파트
OUT       M12142	// R21 H/D1 (IN51) LH 그리퍼 핀 후진확인
; L76
LOAD NOT  P1217F	// R21 H/D1 LH 그리퍼 클램프 잠김1
AND       P12180	// R21 H/D1 LH 그리퍼 클램프 풀림1
AND NOT   P12181	// R21 H/D1 LH 그리퍼 클램프 잠김2
AND       P12182	// R21 H/D1 LH 그리퍼 클램프 풀림2
AND NOT   P12183	// R21 H/D1 LH 그리퍼 클램프 잠김3
AND       P1217E	// R21 H/D1 LH 그리퍼 핀 후진2
OUT       M12143	// R21 H/D1 (IN52) LH 그리퍼 클램프 잠김확인
; L77
LOAD      P1217F	// R21 H/D1 LH 그리퍼 클램프 잠김1
AND NOT   P12180	// R21 H/D1 LH 그리퍼 클램프 풀림1
AND       P12181	// R21 H/D1 LH 그리퍼 클램프 잠김2
AND NOT   P12182	// R21 H/D1 LH 그리퍼 클램프 풀림2
AND       P12183	// R21 H/D1 LH 그리퍼 클램프 잠김3
AND NOT   P1217E	// R21 H/D1 LH 그리퍼 핀 후진2
OUT       M12144	// R21 H/D1 (IN53) LH 그리퍼 클램프 풀림확인
; L78
LOAD      P12184	// R21 H/D1 RH 그리퍼 파트
OUT       M12145	// R21 H/D1 (IN54) RH 그리퍼 파트감지
; L79
LOAD      P12170	// R21 H/D1 RH 그리퍼 핀 전진1
AND NOT   P12171	// R21 H/D1 RH 그리퍼 핀 후진1
AND       P12172	// R21 H/D1 RH 그리퍼 핀 전진2
AND NOT   P12173	// R21 H/D1 RH 그리퍼 핀 후진2
OUT       M12146	// R21 H/D1 (IN55) RH 그리퍼 핀 전진확인
; L80
LOAD NOT  P12170	// R21 H/D1 RH 그리퍼 핀 전진1
AND       P12171	// R21 H/D1 RH 그리퍼 핀 후진1
AND NOT   P12172	// R21 H/D1 RH 그리퍼 핀 전진2
AND       P12173	// R21 H/D1 RH 그리퍼 핀 후진2
OUT       M12147	// R21 H/D1 (IN56) RH 그리퍼 핀 후진확인
; L81
LOAD      P12174	// R21 H/D1 RH 그리퍼 클램프 잠김1
AND NOT   P12175	// R21 H/D1 RH 그리퍼 클램프 풀림1
AND       P12176	// R21 H/D1 RH 그리퍼 클램프 잠김2
AND NOT   P12177	// R21 H/D1 RH 그리퍼 클램프 풀림2
AND       P12178	// R21 H/D1 RH 그리퍼 클램프 잠김3
AND NOT   P12179	// R21 H/D1 RH 그리퍼 클램프 풀림3
OUT       M12148	// R21 H/D1 (IN57) RH 그리퍼 클램프 잠김확인
; L82
LOAD NOT  P12174	// R21 H/D1 RH 그리퍼 클램프 잠김1
AND       P12175	// R21 H/D1 RH 그리퍼 클램프 풀림1
AND NOT   P12176	// R21 H/D1 RH 그리퍼 클램프 잠김2
AND       P12177	// R21 H/D1 RH 그리퍼 클램프 풀림2
AND NOT   P12178	// R21 H/D1 RH 그리퍼 클램프 잠김3
AND       P12179	// R21 H/D1 RH 그리퍼 클램프 풀림3
OUT       M12149	// R21 H/D1 (IN58) RH 그리퍼 클램프 풀림확인
// /////////////////////  그리퍼 제어
; L84
LOAD      P12141	// R21 H/D1 (OT50) LH 그리퍼 핀 전진요구
OUT       M12174	// R21 H/D1 LH 그리퍼 핀 전진 [SOL]

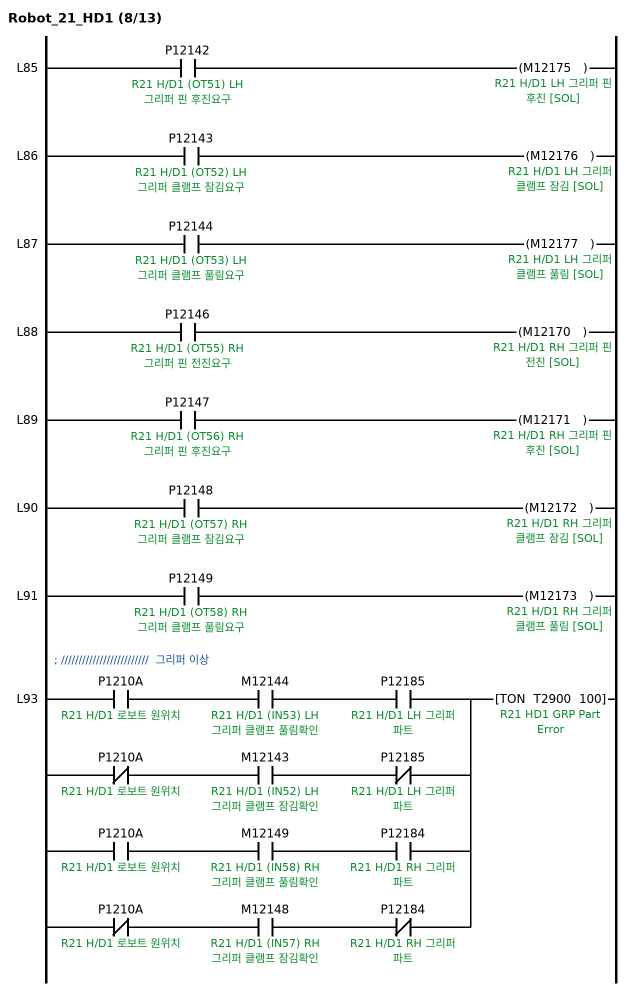
; L85
LOAD      P12142	// R21 H/D1 (OT51) LH 그리퍼 핀 후진요구
OUT       M12175	// R21 H/D1 LH 그리퍼 핀 후진 [SOL]
; L86
LOAD      P12143	// R21 H/D1 (OT52) LH 그리퍼 클램프 잠김요구
OUT       M12176	// R21 H/D1 LH 그리퍼 클램프 잠김 [SOL]
; L87
LOAD      P12144	// R21 H/D1 (OT53) LH 그리퍼 클램프 풀림요구
OUT       M12177	// R21 H/D1 LH 그리퍼 클램프 풀림 [SOL]
; L88
LOAD      P12146	// R21 H/D1 (OT55) RH 그리퍼 핀 전진요구
OUT       M12170	// R21 H/D1 RH 그리퍼 핀 전진 [SOL]
; L89
LOAD      P12147	// R21 H/D1 (OT56) RH 그리퍼 핀 후진요구
OUT       M12171	// R21 H/D1 RH 그리퍼 핀 후진 [SOL]
; L90
LOAD      P12148	// R21 H/D1 (OT57) RH 그리퍼 클램프 잠김요구
OUT       M12172	// R21 H/D1 RH 그리퍼 클램프 잠김 [SOL]
; L91
LOAD      P12149	// R21 H/D1 (OT58) RH 그리퍼 클램프 풀림요구
OUT       M12173	// R21 H/D1 RH 그리퍼 클램프 풀림 [SOL]
// /////////////////////////  그리퍼 이상
; L93
LOAD      P1210A	// R21 H/D1 로보트 원위치
AND       M12144	// R21 H/D1 (IN53) LH 그리퍼 클램프 풀림확인
AND       P12185	// R21 H/D1 LH 그리퍼 파트
LOAD NOT  P1210A	// R21 H/D1 로보트 원위치
AND       M12143	// R21 H/D1 (IN52) LH 그리퍼 클램프 잠김확인
AND NOT   P12185	// R21 H/D1 LH 그리퍼 파트
OR LOAD
LOAD      P1210A	// R21 H/D1 로보트 원위치
AND       M12149	// R21 H/D1 (IN58) RH 그리퍼 클램프 풀림확인
AND       P12184	// R21 H/D1 RH 그리퍼 파트
OR LOAD
LOAD NOT  P1210A	// R21 H/D1 로보트 원위치
AND       M12148	// R21 H/D1 (IN57) RH 그리퍼 클램프 잠김확인
AND NOT   P12184	// R21 H/D1 RH 그리퍼 파트
OR LOAD
TON       T2900 100	// R21 HD1 GRP Part Error 

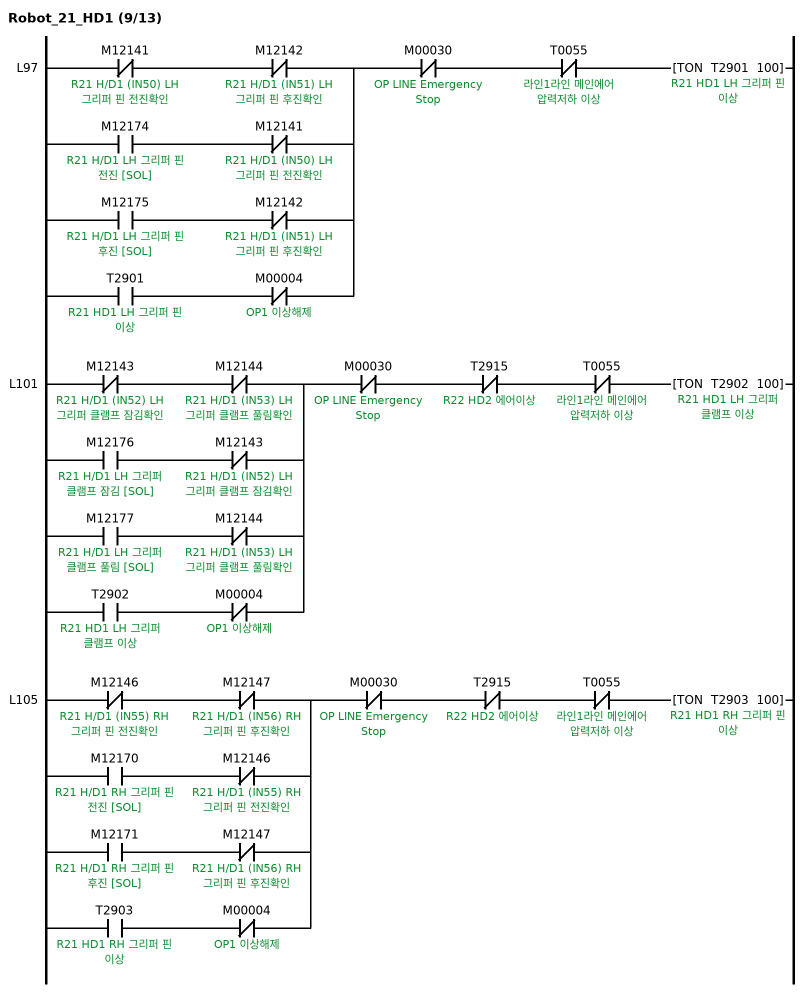
; L97
LOAD NOT  M12141	// R21 H/D1 (IN50) LH 그리퍼 핀 전진확인
AND NOT   M12142	// R21 H/D1 (IN51) LH 그리퍼 핀 후진확인
LOAD      M12174	// R21 H/D1 LH 그리퍼 핀 전진 [SOL]
AND NOT   M12141	// R21 H/D1 (IN50) LH 그리퍼 핀 전진확인
OR LOAD
LOAD      M12175	// R21 H/D1 LH 그리퍼 핀 후진 [SOL]
AND NOT   M12142	// R21 H/D1 (IN51) LH 그리퍼 핀 후진확인
OR LOAD
LOAD      T2901	// R21 HD1 LH 그리퍼 핀 이상
AND NOT   M00004	// OP1 이상해제
OR LOAD
AND NOT   M00030	// OP LINE Emergency Stop
AND NOT   T0055	// 라인1라인 메인에어 압력저하 이상
TON       T2901 100	// R21 HD1 LH 그리퍼 핀 이상
; L101
LOAD NOT  M12143	// R21 H/D1 (IN52) LH 그리퍼 클램프 잠김확인
AND NOT   M12144	// R21 H/D1 (IN53) LH 그리퍼 클램프 풀림확인
LOAD      M12176	// R21 H/D1 LH 그리퍼 클램프 잠김 [SOL]
AND NOT   M12143	// R21 H/D1 (IN52) LH 그리퍼 클램프 잠김확인
OR LOAD
LOAD      M12177	// R21 H/D1 LH 그리퍼 클램프 풀림 [SOL]
AND NOT   M12144	// R21 H/D1 (IN53) LH 그리퍼 클램프 풀림확인
OR LOAD
LOAD      T2902	// R21 HD1 LH 그리퍼 클램프 이상
AND NOT   M00004	// OP1 이상해제
OR LOAD
AND NOT   M00030	// OP LINE Emergency Stop
AND NOT   T2915	// R22 HD2 에어이상
AND NOT   T0055	// 라인1라인 메인에어 압력저하 이상
TON       T2902 100	// R21 HD1 LH 그리퍼 클램프 이상
; L105
LOAD NOT  M12146	// R21 H/D1 (IN55) RH 그리퍼 핀 전진확인
AND NOT   M12147	// R21 H/D1 (IN56) RH 그리퍼 핀 후진확인
LOAD      M12170	// R21 H/D1 RH 그리퍼 핀 전진 [SOL]
AND NOT   M12146	// R21 H/D1 (IN55) RH 그리퍼 핀 전진확인
OR LOAD
LOAD      M12171	// R21 H/D1 RH 그리퍼 핀 후진 [SOL]
AND NOT   M12147	// R21 H/D1 (IN56) RH 그리퍼 핀 후진확인
OR LOAD
LOAD      T2903	// R21 HD1 RH 그리퍼 핀 이상
AND NOT   M00004	// OP1 이상해제
OR LOAD
AND NOT   M00030	// OP LINE Emergency Stop
AND NOT   T2915	// R22 HD2 에어이상
AND NOT   T0055	// 라인1라인 메인에어 압력저하 이상
TON       T2903 100	// R21 HD1 RH 그리퍼 핀 이상

